(* PLC project CoDeSys External Library Template, WAGO e!COCKPIT e!COCKPIT, author 3S - Smart Software Solutions GmbH *)
(* stored: creationDateTime 2019-10-30T07:58:58.440898, version 3.5.5.30, modificationDateTime 2019-10-29T14:38:06.5373783, organization 3S - Smart Software Solutions GmbH *)
(* Library project template with all possible element types, docu and a sample project structure *)

TYPE alARRAYTablicaKomunikatow : ARRAY[1..2000] OF alSTRINGKomunikat;
END_TYPE

TYPE alARRAYTablicaKomunikatowDebug : ARRAY[1..100] OF typKomunikatDebug;
END_TYPE

TYPE alSTRINGjSON : STRING(10000);
END_TYPE

TYPE alSTRINGKomunikat : STRING(1024);
END_TYPE

{attribute 'qualified_only'}
{attribute 'strict'}
TYPE enumAlarmWartosc : (DUPA := 0, StanNormalny := 1, StanAlarmowy := 2);
END_TYPE

(* values of enumKlasaAlarmu: Bezpieczenstwa: najwyższy priorytet alarmu - alarm mogący mieć wpływ na bezpieczeństwo działania budynku; Krytyczny: wysoki priorytet alarmu - alarm istotny mogący doprowadzić do zaistnienia alarmu bezpieczeństwa; Ostrzezenie: średni priorytet alarmu - ostrzeżenie o nieprawidłowym działaniu któregoś z urządzeń; Informacyjny: niski priorytet alarm wyswietlany nie wymagajacy potwierdzenia; AwariaAutomatyki: alarm (podjrzenia) uszkodzenia lub nieprawidłowego działania automatyki; Wewnetrzny: alarm wewnetrzny niewyświetlany nie wymaga potwierdzenia; Systemowy: alarm systemowy niewyświetlany nie wymaga potwierdzenia *)

(* Nazwa bloku: Enumeracja - definicja klasy błędów Projekt: Bałtyckie Centrum Biznesu Budynek 2 Firma: Solwena Autor: Marcin Szumiło Aktualizacja: 2017-11-17-11:00-PK: aktualizacja względem pliku komunikacja 2019-02-13-14:56-AWy: dodanie klasy AwariaAutomatyki *)
{attribute 'qualified_only'}
{attribute 'strict'}
TYPE enumKlasaAlarmu : (Bezpieczenstwa := 0, Krytyczny := 1, Ostrzezenie := 2, Informacyjny := 3, AwariaAutomatyki := 8, Wewnetrzny := 9, Systemowy := 10);
END_TYPE

(* values of enumModbusKodyFunkcji: OdczytWyjscBitowych: odczyt stanu wyjść cyfrowych; OdczytWejscBitowych: odczyt stanu wejść cyfrowych; OdczytNRejestrow: odczyt dowolnej ilości rejestrów; OdczytNRejestrowWejsciowych: odczyt dowolnej ilości rejestrów wejściowych; ZapisBitu: zapis jednego bitu informacji; ZapisRejestru: zapis jednego rejestru; OdczytStatusu: odczyt statusu; ZapisNBitow: zapis dowolnej ilości bitów; ZapisNRejestrow: zapis dowolnej ilości rejestrów *)

(* Nazwa bloku: Enumeracja - definicja kodów funkcyjnych protokołu modbus Projekt: Bałtyckie Centrum Biznesu Budynek 2 Firma: Solwena Autor: Marcin Szumiło Wersja: 0.1.0.1 - 2017-01-10 *)
{attribute 'qualified_only'}
{attribute 'strict'}
TYPE enumModbusKodyFunkcji : (OdczytWyjscBitowych := 1, OdczytWejscBitowych := 2, OdczytNRejestrow := 3, OdczytNRejestrowWejsciowych := 4, ZapisBitu := 5, ZapisRejestru := 6, OdczytStatusu := 7, ZapisNBitow := 15, ZapisNRejestrow := 16);
END_TYPE

(* values of enumModbusStatus: BrakKomunikacji: problem z komunikacją; KomunikacjaPrawidlowa: komunikacja przebiegła prawidłowo *)

(* Nazwa bloku: Enumeracja - definicja kodów błędów w komunikacji modbus Projekt: Bałtyckie Centrum Biznesu Budynek 2 Firma: Solwena Autor: Marcin Szumiło Wersja: 0.1.0.1 - 2017-01-10 *)
{attribute 'qualified_only'}
{attribute 'strict'}
TYPE enumModbusStatus : (BrakKomunikacji := 1, KomunikacjaPrawidlowa := 2);
END_TYPE

(* values of enumPPPSAnalizatorDirisA40Error: BrakKomunikacji: brak komunikacji z analizatorem; BrakZmianyParametrow: alarm braku zmiany wartości paramterów (napięcie, prąd) *)

(* Autor: Paweł Kąkol, 2018-09-04-PK Prawa majątkowe: Solwena Sp. z o.o., Aktualizacje: 2019-02-18-AWy: alarm braku zmiany wartości napięcia lub prądu Opis: fb służy do obsługi alarmów w fb analizatora sieci ECA0 na budynkach PPP Sopot (ENGIE) Diris A40 *)
{attribute 'qualified_only'}
{attribute 'strict'}
TYPE enumPPPSAnalizatorDirisA40Error : (BrakKomunikacji := 1, BrakZmianyParametrow := 2);
END_TYPE

(* Autor: Paweł Kąkol, 2018-09-04-PK Prawa majątkowe: Solwena Sp. z o.o., Aktualizacje: 2019-02-18-AWy: alarm braku zmiany wartości napięcia lub prądu, zmiana klas alarmów Opis: fb służy do definicji klasy alarmów w fb analizatora sieci ECA0 na budynkach PPP Sopot (ENGIE) Diris A40 *)
{attribute 'qualified_only'}
{attribute 'strict'}
TYPE enumPPPSAnalizatorDirisA40ErrorKlasa : (BrakKomunikacji := enumKlasaAlarmu.AwariaAutomatyki, BrakZmianyParametrow := enumKlasaAlarmu.AwariaAutomatyki);
END_TYPE

(* values of enumPPPSBramkaSTC65RS485ModbusError: BrakKomunikacji: brak komunikacji (MODBUS RTU) z konwerterem; ResetKonwertera: reset konwertera; BrakTelegramowEnOcean: brak odbioru telegramów EnOcean (brak komunikacji EnOcean) *)

(* Autor: Paweł Kąkol, 2018-08-13-PK Prawa majątkowe: Solwena Sp. z o.o., Aktualizacje: 2018-09-10-PK - dodanie alarmów ResetKonwertera i BrakTelegramowEnOcean Opis: enum służy do obsługi alarmów w fb konwertera GTW0 na budynkach PPP Sopot *)
{attribute 'qualified_only'}
{attribute 'strict'}
TYPE enumPPPSBramkaSTC65RS485ModbusError : (BrakKomunikacji := 1, ResetKonwertera := 2, BrakTelegramowEnOcean := 3);
END_TYPE

(* Autor: Paweł Kąkol, 2018-08-13-PK Prawa majątkowe: Solwena Sp. z o.o., Aktualizacje: 2018-09-10-PK: dodanie klasy alarmów dla ResetKonwertera i BrakTelegramowEnOcean 2019-02-18-AWy: zmiana klas alarmów Opis: enum służy do definicji klas alarmów w fb konwertera GTW0 na budynkach PPP Sopot *)
{attribute 'qualified_only'}
{attribute 'strict'}
TYPE enumPPPSBramkaSTC65RS485ModbusErrorKlasa : (BrakKomunikacji := enumKlasaAlarmu.AwariaAutomatyki, ResetKonwertera := enumKlasaAlarmu.AwariaAutomatyki, BrakTelegramowEnOcean := enumKlasaAlarmu.AwariaAutomatyki);
END_TYPE

(* values of enumPPPSDestratyfikatorTBOXError: BrakKomunikacji: brak komunikacji z węzłem; AlarmCzujnika: alarm braku zmiany wartości czujnika temp. *)

(* Autor: Artur Wyszomirski, 2019-02-05-AWy Prawa majątkowe: Solwena Sp. z o.o., Aktualizacje: 2019-02-18-AWy - alarm czujnika temperatury Opis: enum służy do obsługi alarmów w fb węzła Frisko ATTOM1S na budynkach PPP Sopot (ENGIE) *)
{attribute 'qualified_only'}
{attribute 'strict'}
TYPE enumPPPSDestratyfikatorTBOXError : (BrakKomunikacji := 1, AlarmCzujnika := 2);
END_TYPE

(* Autor: Paweł Kąkol, 2018-09-03-PK Prawa majątkowe: Solwena Sp. z o.o., Aktualizacje: 2019-02-18-AWy: alarm czujnika temperatury 2019-02-18-AWy: zmiana klas alarmów Opis: enum służy do definicji klas alarmów w fb węzła Climatix POL63x na budynkach PPP Sopot (ENGIE) *)
{attribute 'qualified_only'}
{attribute 'strict'}
TYPE enumPPPSDestratyfikatorTBOXErrorKlasa : (BrakKomunikacji := enumKlasaAlarmu.AwariaAutomatyki, AlarmCzujnika := enumKlasaAlarmu.AwariaAutomatyki);
END_TYPE

(* values of enumPPPSFriskoATTOM1SError: BrakKomunikacji: brak komunikacji z węzłem; AlarmCzujnikaZewnetrznego: alarm braku zmiany wartości czujnika temp. zewnetrznj; AlarmCzujnikaZasilaniaObwoduCO: alarm braku zmiany wartości czujnika temp. zasilana obwod c. o.; BrakOsiagnieciaTemperaturyCO: alarm braku osiągnięcia temp. zadanej obwodu c. o.; BladIloscPomiarowTemperatury: alarm zbyt małej ilości pomiarów dokonanych w ciągu dnia do obliczenia średniej *)

(* Autor: Artur Wyszomirski, 2019-02-05-AWy Prawa majątkowe: Solwena Sp. z o.o., Aktualizacje: 2019-02-19-AWy: dodanie alarmów czujnika zew., zasilania c.o., braku osiągnięcia temperatury zadanej Opis: enum służy do obsługi alarmów w fb węzła Frisko ATTOM1S na budynkach PPP Sopot (ENGIE) *)
{attribute 'qualified_only'}
{attribute 'strict'}
TYPE enumPPPSFriskoATTOM1SError : (BrakKomunikacji := 1, AlarmCzujnikaZewnetrznego := 2, AlarmCzujnikaZasilaniaObwoduCO := 3, BrakOsiagnieciaTemperaturyCO := 4, BladIloscPomiarowTemperatury := 5);
END_TYPE

(* values of enumPPPSFriskoATTOM1SErrorKlasa: AlarmCzujnikaZewnetrznego: alarm braku zmiany wartości czujnika temp. zewnetrznj; AlarmCzujnikaZasilaniaObwoduCO: alarm braku zmiany wartości czujnika temp. zasilana obwod c. o.; BrakOsiagnieciaTemperaturyCO: alarm braku osiągnięcia temp. zadanej obwodu c. o.; BladIloscPomiarowTemperatury: alarm zbyt małej ilości pomiarów dokonanych w ciągu dnia do obliczenia średniej *)

(* Autor: Paweł Kąkol, 2018-09-03-PK Prawa majątkowe: Solwena Sp. z o.o., Aktualizacje: 2019-02-19-AWy: dodanie alarmów czujnika zew., zasilania c.o., braku osiągnięcia temperatury zadanej 2019-02-18-AWy: zmiana klas alarmów Opis: enum służy do definicji klas alarmów w fb węzła Climatix POL63x na budynkach PPP Sopot (ENGIE) *)
{attribute 'qualified_only'}
{attribute 'strict'}
TYPE enumPPPSFriskoATTOM1SErrorKlasa : (BrakKomunikacji := enumKlasaAlarmu.AwariaAutomatyki, AlarmCzujnikaZewnetrznego := enumKlasaAlarmu.AwariaAutomatyki, AlarmCzujnikaZasilaniaObwoduCO := enumKlasaAlarmu.AwariaAutomatyki, BrakOsiagnieciaTemperaturyCO := enumKlasaAlarmu.Ostrzezenie, BladIloscPomiarowTemperatury := enumKlasaAlarmu.AwariaAutomatyki);
END_TYPE

(* values of enumPPPSFriskoATTOM1STrybPracy: Zima: Zima; Lato: Lato; Auto: Automatyczny - przełączenie trybów uzależnione od temperatury zewnętrznej *)

(* Autor: Artur Wyszomirski, 22.05.2019 Prawa majątkowe: Solwena Sp. z o.o., Aktualizacje: Opis: enum służy do obsługi Trybów pracy fb węzła Frisko ATTO M1S na budynkach PPP Sopot (ENGIE) *)
{attribute 'qualified_only'}
{attribute 'strict'}
TYPE enumPPPSFriskoATTOM1STrybPracy : (Zima := 0, Lato := 1, Auto := 2);
END_TYPE

(* values of enumPPPSHarmonogramy: Ekonomiczny: Tryb pracy ekonomicznej; Komfort: Tryb pracy komfortu *)

(* Autor: Paweł Kąkol, 2018-09-10-PK Prawa majątkowe: Solwena Sp. z o.o., Aktualizacje: Opis: enum służy do obsługi Trybów pracy harmonogramu na budynkach PPP Sopot (ENGIE) *)
{attribute 'qualified_only'}
{attribute 'strict'}
TYPE enumPPPSHarmonogramy : (Ekonomiczny := 0, Komfort := 1);
END_TYPE

(* values of enumPPPSKlimatyzatorTroxSchoolairVError: BrakKomunikacji: brak komunikacji z węzłem; AlarmCzujnika: alarm braku zmiany wartości czujnika temp. *)

(* Autor: Artur Wyszomirski, 2019-02-05-AWy Prawa majątkowe: Solwena Sp. z o.o., Aktualizacje: 2019-02-18-AWy - alarm czujnika temperatury Opis: enum służy do obsługi alarmów w fb węzła Frisko ATTOM1S na budynkach PPP Sopot (ENGIE) *)
{attribute 'qualified_only'}
{attribute 'strict'}
TYPE enumPPPSKlimatyzatorTroxSchoolairVError : (BrakKomunikacji := 1, AlarmCzujnika := 2);
END_TYPE

(* Autor: Paweł Kąkol, 2018-09-03-PK Prawa majątkowe: Solwena Sp. z o.o., Aktualizacje: 2019-02-18-AWy: alarm czujnika temperatury 2019-02-18-AWy: zmiana klas alarmów Opis: enum służy do definicji klas alarmów w fb węzła Climatix POL63x na budynkach PPP Sopot (ENGIE) *)
{attribute 'qualified_only'}
{attribute 'strict'}
TYPE enumPPPSKlimatyzatorTroxSchoolairVErrorKlasa : (BrakKomunikacji := enumKlasaAlarmu.AwariaAutomatyki, AlarmCzujnika := enumKlasaAlarmu.AwariaAutomatyki);
END_TYPE

(* values of enumPPPSLicznikCieplaMultical403Error: BrakKomunikacji: Brak komunikacji z węzłem; AlarmCzujnikaPrzeplywu: Alarm braku zmiany wartości czujnika przepływu; AlarmCzujnikaZasilania: Alarm braku zmiany wartości czujnika temp. zasilania; AlarmCzujnikaPowrotu: Alarm braku zmiany wartości czujnika temp. powrotu *)

(* Autor: Artur Wyszomirski, 2019-08-07-AWy Prawa majątkowe: Solwena Sp. z o.o., Aktualizacje: Opis: Enumeracja alarmów w fb licznia ciepła Multical403 *)
{attribute 'qualified_only'}
{attribute 'strict'}
TYPE enumPPPSLicznikCieplaMultical403Error : (BrakKomunikacji := 1, AlarmCzujnikaPrzeplywu := 2, AlarmCzujnikaZasilania := 3, AlarmCzujnikaPowrotu := 4);
END_TYPE

(* values of enumPPPSLicznikCieplaMultical403ErrorKlasa: AlarmCzujnikaPrzeplywu: Alarm braku zmiany wartości czujnika przepływu; AlarmCzujnikaZasilania: Alarm braku zmiany wartości czujnika temp. zasilania; AlarmCzujnikaPowrotu: Alarm braku zmiany wartości czujnika temp. powrotu *)

(* Autor: Artur Wyszomirski, 2019-08-07-AWy Prawa majątkowe: Solwena Sp. z o.o., Aktualizacje: Opis: Klasy alarmów w fb licznia ciepła Multical403 *)
{attribute 'qualified_only'}
{attribute 'strict'}
TYPE enumPPPSLicznikCieplaMultical403ErrorKlasa : (BrakKomunikacji := enumKlasaAlarmu.AwariaAutomatyki, AlarmCzujnikaPrzeplywu := enumKlasaAlarmu.AwariaAutomatyki, AlarmCzujnikaZasilania := enumKlasaAlarmu.AwariaAutomatyki, AlarmCzujnikaPowrotu := enumKlasaAlarmu.Ostrzezenie);
END_TYPE

(* values of enumPPPSLicznikCieplaMultical602Error: BrakKomunikacji: Brak komunikacji z węzłem; AlarmCzujnikaPrzeplywu: Alarm braku zmiany wartości czujnika przepływu; AlarmCzujnikaZasilania: Alarm braku zmiany wartości czujnika temp. zasilania; AlarmCzujnikaPowrotu: Alarm braku zmiany wartości czujnika temp. powrotu *)

(* Autor: Artur Wyszomirski, 2019-08-08-AWy Prawa majątkowe: Solwena Sp. z o.o., Aktualizacje: Opis: Enumeracja alarmów w fb licznia ciepła Multical602 *)
{attribute 'qualified_only'}
{attribute 'strict'}
TYPE enumPPPSLicznikCieplaMultical602Error : (BrakKomunikacji := 1, AlarmCzujnikaPrzeplywu := 2, AlarmCzujnikaZasilania := 3, AlarmCzujnikaPowrotu := 4);
END_TYPE

(* values of enumPPPSLicznikCieplaMultical602ErrorKlasa: AlarmCzujnikaPrzeplywu: Alarm braku zmiany wartości czujnika przepływu; AlarmCzujnikaZasilania: Alarm braku zmiany wartości czujnika temp. zasilania; AlarmCzujnikaPowrotu: Alarm braku zmiany wartości czujnika temp. powrotu *)

(* Autor: Artur Wyszomirski, 2019-08-08-AWy Prawa majątkowe: Solwena Sp. z o.o., Aktualizacje: Opis: Klasy alarmów w fb licznia ciepła Multical602 *)
{attribute 'qualified_only'}
{attribute 'strict'}
TYPE enumPPPSLicznikCieplaMultical602ErrorKlasa : (BrakKomunikacji := enumKlasaAlarmu.AwariaAutomatyki, AlarmCzujnikaPrzeplywu := enumKlasaAlarmu.AwariaAutomatyki, AlarmCzujnikaZasilania := enumKlasaAlarmu.AwariaAutomatyki, AlarmCzujnikaPowrotu := enumKlasaAlarmu.Ostrzezenie);
END_TYPE

(* values of enumPPPSPomieszczenie: SalaLekcyjna: Sale lekcyjne, przedszkolne, świetlica, biblioteka (20 st. C); SalaNiemowlat: Sale niemowląt, dziecięce w żłobkach (24 st. C); Rehabilitacyjne: Pomieszczenia rehabilitacyjne SPON (24 st. C); Korytarz: Korytarze (20 st. C); Szatnia: Szatnie (16 st. C); SalaGimnastyczna: Sale gimnastyczne (16 st. C); Lazienka: Łazienki i ustępy (24 st. C); PomieszczenieBiurowe: Pomieszczenia biurowe i administracyjne (20 st. C); PomieszczenieMieszkalne: Pomieszczenia mieszkalne, przedpokoje, kuchnie (20 st. C); Magazyn: Pomieszczenia magazynowe (16 st. C) *)

(* Autor: Artur Wyszomirski, 2018-10-15-AW; Prawa majątkowe: Solwena Sp. z o.o., Aktualizacje: Opis: enum służy do obsługi rodzajów pomieszczeń w budynkach PPP Sopot (ENGIE) *)
{attribute 'qualified_only'}
{attribute 'strict'}
TYPE enumPPPSPomieszczenie : (SalaLekcyjna := 0, SalaNiemowlat := 1, Rehabilitacyjne := 2, Korytarz := 3, Szatnia := 4, SalaGimnastyczna := 5, Lazienka := 6, PomieszczenieBiurowe := 7, PomieszczenieMieszkalne := 8, Magazyn := 9);
END_TYPE

(* values of enumPPPSSilownikSABpError: BrakKomunikacji: brak komunikacji (po EnOcean) z siłownikiem; AlarmOgolny: alarm ogólny; DetekcjaOtwarciaOkna: błąd baterii; Defrost: defrost; AlarmCzujnika: alarm braku zmiany wartości czujnika temp. *)

(* Autor: Paweł Kąkol, 2018-09-04-PK Prawa majątkowe: Solwena Sp. z o.o., Aktualizacje: 2019-01-28-JC - defrost 2019-02-14-AWy - alarm czujnika temperatury Opis: enum służy do obsługi alarmów w fb siłownika (SAB+) HRU0 na budynkach PPP Sopot *)
{attribute 'qualified_only'}
{attribute 'strict'}
TYPE enumPPPSSilownikSABpError : (BrakKomunikacji := 1, AlarmOgolny := 2, DetekcjaOtwarciaOkna := 3, Defrost := 4, AlarmCzujnika := 5);
END_TYPE

(* Autor: Paweł Kąkol, 2018-09-04-PK Prawa majątkowe: Solwena Sp. z o.o., Aktualizacje: 2019-01-28-JC: defrost 2019-02-14-AWy: alarm czujnika temperatury 2019-02-18-AWy: zmiana klas alarmów Opis: enum służy do definicji klas alarmów w fb siłownika (SAB+) HRU0 na budynkach PPP Sopot *)
{attribute 'qualified_only'}
{attribute 'strict'}
TYPE enumPPPSSilownikSABpErrorKlasa : (BrakKomunikacji := enumKlasaAlarmu.AwariaAutomatyki, AlarmOgolny := enumKlasaAlarmu.Ostrzezenie, DetekcjaOtwarciaOkna := enumKlasaAlarmu.Informacyjny, Defrost := enumKlasaAlarmu.Bezpieczenstwa, AlarmCzujnika := enumKlasaAlarmu.AwariaAutomatyki);
END_TYPE

(* values of enumPPPSSilownikSABpServiceFlag: BrakDzialan: Brak rozkazu; TrybLetni: Rozkaz ustwienia trybu letniego; ZamkniecieZaworu: Rozkaz zamknięcia zaworu; OtwarcieZaworu: Rozkaz otwarcia zaworu; PozycjaGorna: Rozkaz pozycji górnej trzpienia (pozycja do transportu) - po jego uruchomieniu wymagana ponowna kalibracja; KalibracjaSilownika: Rozkaz uruchomienia sekwencji inicjalizacji siłownika *)

(* Autor: Paweł Kąkol, 2018-09-04-PK Prawa majątkowe: Solwena Sp. z o.o., Aktualizacje: Opis: enum służy do obsługi flagi serwisowej siłownika SAB+ (HRU0) na budynkach PPP Sopot (ENGIE) *)
{attribute 'qualified_only'}
{attribute 'strict'}
TYPE enumPPPSSilownikSABpServiceFlag : (BrakDzialan := 0, TrybLetni := 1, ZamkniecieZaworu := 2, OtwarcieZaworu := 3, PozycjaGorna := 4, KalibracjaSilownika := 5);
END_TYPE

(* values of enumPPPSSilownikTrybPracy: Manualny: Tryb pracy ręcznej; Automatyczny: Tryb pracy automatycznej *)

(* Autor: Artur Wyszomirski, 2018-09-25-AW Prawa majątkowe: Solwena Sp. z o.o., Aktualizacje: Opis: enum służy do obsługi Trybów pracy fb siłownika SABp (HRU0) na budynkach PPP Sopot (ENGIE) *)
{attribute 'qualified_only'}
{attribute 'strict'}
TYPE enumPPPSSilownikTrybPracy : (Manualny := 0, Automatyczny := 1);
END_TYPE

{attribute 'qualified_only'}
{attribute 'strict'}
TYPE enumPPPSUrzadenieStatus : (Nieaktywny := 1, Oczekiwanie := 2, Prawidlowy := 3, Ostrzezenie := 4, Awaria := 5, Krytyczny := 6);
END_TYPE

(* values of enumPPPSWezelClimatixPOL63xError: BrakKomunikacji: brak komunikacji z zadajnikiem; AlarmOgolnyBezpieczenstwa: alarm ogólny bezpieczeństwa; AlarmOgolnyKrytyczny: alarm ogólny krytyczny; AlarmOgolnyOstrzezenie: alarm ogólny ostrzeżenie; AlarmOgolnyInformacyjny: alarm ogólny informacyjny; AlarmCzujnikaZewnetrznego: alarm braku zmiany wartości czujnika temp. zewnetrznj; AlarmCzujnikaZasilaniaObwoduHC1: alarm braku zmiany wartości czujnika temp. zasilana obwodu HC1; AlarmCzujnikaZasilaniaObwoduDHW: alarm braku zmiany wartości czujnika temp. zasilana obwodu DHW; AlarmBrakuOsiagnieciaTemperaturyHC1: alarm braku osiągnięcia temp. zadanej obwodu HC1; AlarmBrakuOsiagnieciaTemperaturyDHW: alarm braku osiągnięcia temp. zadanej obwodu DHW; BladIloscPomiarowTemperatury: alarm zbyt małej ilości pomiarów dokonanych w ciągu dnia do obliczenia średniej *)

(* Autor: Paweł Kąkol, 2018-09-03-PK Prawa majątkowe: Solwena Sp. z o.o., Aktualizacje: 2019-02-14-AWy: dodanie alarmów czujników temp. zewnętrznej i zasilania obwodu HC1, DHW Opis: enum służy do obsługi alarmów w fb węzła Climatix POL63x na budynkach PPP Sopot (ENGIE) *)
{attribute 'qualified_only'}
{attribute 'strict'}
TYPE enumPPPSWezelClimatixPOL63xError : (BrakKomunikacji := 1, AlarmOgolnyBezpieczenstwa := 2, AlarmOgolnyKrytyczny := 3, AlarmOgolnyOstrzezenie := 4, AlarmOgolnyInformacyjny := 5, AlarmCzujnikaZewnetrznego := 6, AlarmCzujnikaZasilaniaObwoduHC1 := 7, AlarmCzujnikaZasilaniaObwoduDHW := 8, AlarmBrakuOsiagnieciaTemperaturyHC1 := 9, AlarmBrakuOsiagnieciaTemperaturyDHW := 10, BladIloscPomiarowTemperatury := 11);
END_TYPE

(* values of enumPPPSWezelClimatixPOL63xErrorKlasa: AlarmCzujnikaZewnetrznego: alarm braku zmiany wartości czujnika temp. zewnetrznj; AlarmCzujnikaZasilaniaObwoduHC1: alarm braku zmiany wartości czujnika temp. zasilana obwodu HC1; AlarmCzujnikaZasilaniaObwoduDHW: alarm braku zmiany wartości czujnika temp. zasilana obwodu DHW; AlarmBrakuOsiagnieciaTemperaturyHC1: alarm braku osiągnięcia temp. zadanej obwodu HC1; AlarmBrakuOsiagnieciaTemperaturyDHW: alarm braku osiągnięcia temp. zadanej obwodu DHW; BladIloscPomiarowTemperatury: alarm zbyt małej ilości pomiarów dokonanych w ciągu dnia do obliczenia średniej *)

(* Autor: Paweł Kąkol, 2018-09-03-PK Prawa majątkowe: Solwena Sp. z o.o., Aktualizacje: 2019-02-14-AWy: dodanie alarmów czujników temp. zewnętrznej i zasilania obwodu HC1, DHW 2019-02-18-AWy: zmiana klas alarmów Opis: enum służy do definicji klas alarmów w fb węzła Climatix POL63x na budynkach PPP Sopot (ENGIE) *)
{attribute 'qualified_only'}
{attribute 'strict'}
TYPE enumPPPSWezelClimatixPOL63xErrorKlasa : (BrakKomunikacji := enumKlasaAlarmu.AwariaAutomatyki, AlarmOgolnyBezpieczenstwa := enumKlasaAlarmu.Bezpieczenstwa, AlarmOgolnyKrytyczny := enumKlasaAlarmu.Krytyczny, AlarmOgolnyOstrzezenie := enumKlasaAlarmu.Ostrzezenie, AlarmOgolnyInformacyjny := enumKlasaAlarmu.Informacyjny, AlarmCzujnikaZewnetrznego := enumKlasaAlarmu.AwariaAutomatyki, AlarmCzujnikaZasilaniaObwoduHC1 := enumKlasaAlarmu.AwariaAutomatyki, AlarmCzujnikaZasilaniaObwoduDHW := enumKlasaAlarmu.AwariaAutomatyki, AlarmBrakuOsiagnieciaTemperaturyHC1 := enumKlasaAlarmu.Ostrzezenie, AlarmBrakuOsiagnieciaTemperaturyDHW := enumKlasaAlarmu.Ostrzezenie, BladIloscPomiarowTemperatury := enumKlasaAlarmu.AwariaAutomatyki);
END_TYPE

(* values of enumPPPSWezelClimatixPOL63xTrybPracy: Auto: Tryb pracy automatycznej; OchronaBudynku: Tryb utrzymania minimalnych nastaw dla ochrony budynku; Ekonomiczny: Tryb Ekonomiczny; Komfort: Tryb komfortu; ReczneWylaczenie: Ręczne, lokalne wyłączenie węzła *)

(* Autor: Paweł Kąkol, 2018-09-03-PK Prawa majątkowe: Solwena Sp. z o.o., Aktualizacje: Opis: enum służy do obsługi Trybów pracy fb węzła Climatix POL63x na budynkach PPP Sopot (ENGIE) *)
{attribute 'qualified_only'}
{attribute 'strict'}
TYPE enumPPPSWezelClimatixPOL63xTrybPracy : (Auto := 0, OchronaBudynku := 1, Ekonomiczny := 2, Komfort := 3, ReczneWylaczenie := 4);
END_TYPE

(* values of enumPPPSZadajnikError: BrakKomunikacji: brak komunikacji z zadajnikiem (po EnOcean); AlarmOgolny: alarm ogólny; AlarmCzujnika: alarm braku zmiany wartości czujnika temp. *)

(* Autor: Paweł Kąkol, 2018-08-13-PK Prawa majątkowe: Solwena Sp. z o.o., Aktualizacje: 2019-02-14-AWy - alarm czujnika temperatury Opis: enum służy do obsługi alarmów w fb zadajnika FCP0 na budynkach PPP Sopot *)
{attribute 'qualified_only'}
{attribute 'strict'}
TYPE enumPPPSZadajnikError : (BrakKomunikacji := 1, AlarmOgolny := 2, AlarmCzujnika := 3);
END_TYPE

(* Autor: Paweł Kąkol, 2018-08-13-PK Prawa majątkowe: Solwena Sp. z o.o., Aktualizacje: 2019-02-14-AWy: alarm czujnika temperatury 2019-02-18-AWy: zmiana klas alarmów Opis: enum służy do definicji klas alarmów w fb zadajnika FCP0 na budynkach PPP Sopot *)
{attribute 'qualified_only'}
{attribute 'strict'}
TYPE enumPPPSZadajnikErrorKlasa : (BrakKomunikacji := enumKlasaAlarmu.AwariaAutomatyki, AlarmOgolny := enumKlasaAlarmu.Ostrzezenie, AlarmCzujnika := enumKlasaAlarmu.AwariaAutomatyki);
END_TYPE

(* values of enumPPPSZadajnikTrybPracy: Manualny: Tryb pracy ręcznej; Automatyczny: Tryb pracy automatyczny *)

(* Autor: Paweł Kąkol, 2018-09-10-PK Prawa majątkowe: Solwena Sp. z o.o., Aktualizacje: 2018-10-02 - AW - Zmiana numeracji. Tryb Manualny na 0 2018-10-15 - AW - Zmiana numeracji. Dodanie trybów AutonomizacjaManualny i AutonomizacjaAutomatyczny 2018-12-12 - JB - Ujednolicenie trybów z siłownikiem SAB+. 2019-06-06 - AWy - Usunięcie trybów Wylaczenie, AutonomizacjaManualny i AutonomizacjaAutomatyczny oraz zmiana nazwy trybu Regulacja IZE na Automatyczny Opis: enum służy do obsługi Trybów pracy fb zadajnika SR04P (FCP0) na budynkach PPP Sopot (ENGIE) *)
{attribute 'qualified_only'}
{attribute 'strict'}
TYPE enumPPPSZadajnikTrybPracy : (Manualny := 0, Automatyczny := 1);
END_TYPE

{attribute 'qualified_only'}
{attribute 'strict'}
TYPE enumSystemError : (BrakHeartbetuzIZE := 1, NiezgodnaIloscKomunikatowOdebranychZIZE := 2, BladCRCWKomunikacieZIZE := 3, BladSzyfrowania := 4, ZaDuzaIloscKomunikatowWBuforze := 5, BladWalidacjiFullIdentifier := 6, BladFullIdentifierWHeartBeat := 7, BlokadaWysylaniaRamek := 8);
END_TYPE

{attribute 'qualified_only'}
{attribute 'strict'}
TYPE enumSystemErrorKlasa : (BrakHeartbetuzIZE := enumKlasaAlarmu.Krytyczny, NiezgodnaIloscKomunikatowOdebranychZIZE := enumKlasaAlarmu.Systemowy, BladCRCWKomunikacieZIZE := enumKlasaAlarmu.Systemowy, BladSzyfrowania := enumKlasaAlarmu.Systemowy, ZaDuzaIloscKomunikatowWBuforze := enumKlasaAlarmu.Systemowy, BladWalidacjiFullIdentifier := enumKlasaAlarmu.Systemowy, BladFullIdentifierWHeartBeat := enumKlasaAlarmu.Systemowy, BlokadaWysylaniaRamek := enumKlasaAlarmu.Systemowy);
END_TYPE

TYPE SILOWNIK_HRU : STRUCT
  sIdInstancji : STRING;
  intTrybPracy : INT;
  xBrakKomunikacjiIZE : BOOL;
  xBrakKomunikacjiPLC : BOOL;
  xPokazPanelHMI : BOOL := TRUE;
  rTemperaturaPomieszczenia : REAL;
  rNastawaPolozeniaSilownika : REAL;
  rZadanePolozenieSilownikaHMI : REAL;
  intTrybPracyHMI : INT := 1;
  xAutonomizacja : BOOL;
  xAlarmOgolny : BOOL;
  xBladBaterii : BOOL;
  xDetekcjaOtwarciaOkna : BOOL;
  sEnOceanIDodczytany : STRING;
  wCzasOdOstatniegoKomunikatu : WORD;
  xPoprawneParowanie : BOOL;
  xUczenieWlaczHMI : BOOL;
  xUczenieWlaczone : BOOL;
  xUsuwaniePotwierdzenieHMI : BOOL;
  xUsuwanieHMI : BOOL;
END_STRUCT;
END_TYPE

TYPE STEROWNIK_LAC : STRUCT
  xAutonomizacjaWyjscie : BOOL;
END_STRUCT;
END_TYPE

TYPE typHarmonogramDzien : STRUCT
  uintDzienTygodnia : UINT;
  arZdarzenia : ARRAY[0..24] OF typHarmonogramZdarzenie;
END_STRUCT;
END_TYPE

TYPE typHarmonogramJSON : STRUCT
  sPokoj : STRING(3);
  sPietro : STRING(2);
  arHarmonogramTygodniowy : ARRAY[0..6] OF typHarmonogramDzien;
  arWyjatki : ARRAY[0..24] OF typHarmonogramWyjatek;
END_STRUCT;
END_TYPE

TYPE typHarmonogramWyjatek : STRUCT
  dData : DATE;
  arZdarzenia : ARRAY[0..9] OF typHarmonogramZdarzenie;
END_STRUCT;
END_TYPE

TYPE typHarmonogramZdarzenie : STRUCT
  dtCzasRozpoczecia : DT;
  dtCzasZakonczenia : DT;
  sNazwaAtrybutu : STRING(15);
  sWartoscAtrybutu : STRING(15);
END_STRUCT;
END_TYPE

TYPE typKomunikat : STRUCT
  sZnacznik : STRING;
  sTypKomunikatu : STRING;
  sMnemonikWlasciciela : STRING;
  sMnemonikWlascicielaExt : STRING;
  sMACAdres : STRING;
  sIDZrodla : STRING;
  sIDZrodlaLokalizacja : STRING;
  sIDZrodlaUrzadzenie : STRING;
  sIDPrzeznaczenia : STRING;
  sIDPrzeznaczeniaLokalizacja : STRING;
  sIDPrzeznaczeniaUrzadzenie : STRING;
  sDlugoscPolaDanych : STRING;
  sMarkerCzasowy : STRING;
  sRezerwa : STRING;
  sDane : alSTRINGKomunikat;
END_STRUCT;
END_TYPE

TYPE typKomunikatDebug : STRUCT
  intGlobalnyZnacznikWysylkiUDP : INT;
  intGlobalnyZnacznikOdczytu : INT;
  intGlobalnyZnacznikZapisu : INT;
  intGlobalnaLiczbaKomunikatowWBuforze : INT;
  dtLokalnyCzasSterownika : DT;
  sDane : alSTRINGKomunikat;
END_STRUCT;
END_TYPE

TYPE typModbusOdczytCykliczny : STRUCT
  bAdresUrzadzenia : BYTE;  (* ID urządzenia SLAVE w sieci MODBUS *)
  bFunkcja : BYTE;  (* kod funkcji użytej w rozkazie MODBUS *)
  uiAdresRejestru : UINT;  (* rejestr startowy *)
  ltCzestotliwosc : LTIME;  (* po jakim czasie w ms ma być wysłany następny request *)
  ltZnacznikCzasuWyslania : LTIME;  (* znacznik czasowy próby wykonania rozkazu *)
  pZmiennaReferencyjna : POINTER TO WORD;  (* wskaźnik do zmiennej INT przechowującej wynik *)
END_STRUCT;
END_TYPE

TYPE typModbusOdczytZapisZadanie : STRUCT
  bAdresUrzadzenia : BYTE;  (* ID urządzenia SLAVE w sieci MODBUS *)
  bFunkcja : BYTE;  (* kod funkcji użytej w rozkazie MODBUS *)
  uiAdresRejestru : UINT;  (* rejestr startowy *)
  pZmiennaDoOdczytu : POINTER TO WORD;  (* wskaźnik do zmiennej INT przechowującej wynik *)
  wWartoscDoZapisania : WORD;  (* wartość do zapisania *)
END_STRUCT;
END_TYPE

TYPE typModbusRTUParametryKomunikacji : STRUCT
  xKomunikacjaAktywna : BOOL;
  typNazwaPortuKomunikacyjnego : WagoTypesCom.I_WagoSysComBase;
  udiPredkosc : UDINT;
  usiBityDanych : USINT;
  eParzystosc : eTTYParity;
  eBityStopu : eTTYStopBits;
  eHandshake : eTTYHandshake;
  eDuplex : eTTYPhysicalLayer;
  eTypRamki : eMbFrameType;
  tTimeout : TIME;
END_STRUCT;
END_TYPE

TYPE typModbusTCPParametryKomunikacji : STRUCT
  xKomunikacjaAktywna : BOOL;
  sAdresTCP : STRING;
  wPortTCP : WORD;
  utPodtrzymajWtyczkeTCP : typKeepAlive;
  eTypRamki : eMbFrameType;
  tTimeOut : TIME;
END_STRUCT;
END_TYPE

TYPE typWirtualnePomieszczenie : STRUCT
  sIDPomieszczenia : STRING;
  intObecnosc : INT := -1;
END_STRUCT;
END_TYPE

TYPE ZADAJNIK_FCP : STRUCT
  sIdInstancji : STRING;
  rTemperaturaNastawiona : REAL;
  rTemperaturaPomieszczenia : REAL;
  rTemperaturaBazowaHMI : REAL := 293.15;
  rSkalaPotencjometruAutonomizacja : REAL := 1;
  rTemperaturaBazowaAutoAutonomizacja : REAL := 293.15;
  intTrybPracy : INT;
  xBrakKomunikacjiIZE : BOOL;
  xBrakKomunikacjiPLC : BOOL;
  xPokazPanelHMI : BOOL := TRUE;
  intTrybPracyHMI : INT := 1;
  xAutonomizacja : BOOL;
  sEnOceanIDodczytany : STRING;
  wCzasOdOstatniegoKomunikatu : WORD;
  xZwiekszTemperature : BOOL;
  xZmniejszTemperature : BOOL;
END_STRUCT;
END_TYPE

(* Nazwa bloku: Blok funkcyjny konwersji liczby decymalnej na binarną Autor: Jan Bartczak Wersja: v1.0.0 - 2018-06-22 *)
FUNCTION_BLOCK fbDecToBin
  VAR_INPUT
    wWordWejsciowy : WORD;
    intIloscBitow : INT;
  END_VAR
  VAR_OUTPUT
    arBity : ARRAY[0..16] OF BYTE;
  END_VAR
  VAR
    intWejsciowy : UINT;
    bBajtPojedynczy : BYTE;
    intWord : WORD;
    intI : INT;
  END_VAR

            intWejsciowy := WORD_TO_UINT(wWordWejsciowy);
intIloscBitow := intIloscBitow - 1;
FOR intI := 0 TO intIloscBitow BY 1 DO
	intWord := (intWejsciowy MOD 2);
	bBajtPojedynczy := UINT_TO_BYTE(intWord);
	arBity[intI] := bBajtPojedynczy;
	intWejsciowy := intWejsciowy/2;
END_FOR;

          
END_FUNCTION_BLOCK

FUNCTION_BLOCK fbFiltrWartoscAnalogowa
  VAR_INPUT
    rWartoscWejsciowa : REAL;
    rWartoscWejsciowaZaraportowana : REAL;
    rDeadband : REAL;
    tCzasMinimalny : TIME := TIME#5s0ms;
    tCzasMaksymalny : TIME := TIME#1m0s0ms;
    rWynikMnoznik : REAL := 1;
    rWynikOffset : REAL := 0;
  END_VAR
  VAR_OUTPUT
    rWartoscWyjsciowa : REAL;
  END_VAR
  VAR
    rWartoscWejsciowaZaraportowanaReferencja : REAL;
    fbCzasMinimalny : TON;
    fbCzasMaksymalny : TON;
    xCzasMinimalny : BOOL;
    xCzasMaksymalny : BOOL;
  END_VAR

            xCzasMinimalny := TRUE;
xCzasMaksymalny := TRUE;	

IF rWartoscWejsciowaZaraportowana <> rWartoscWejsciowaZaraportowanaReferencja THEN
	rWartoscWejsciowaZaraportowanaReferencja := rWartoscWejsciowaZaraportowana;
	xCzasMinimalny := FALSE;
	xCzasMaksymalny := FALSE;	
END_IF

IF fbCzasMinimalny.Q AND ABS(rWartoscWyjsciowa - (rWartoscWejsciowa * rWynikMnoznik + rWynikOffset)) > rDeadband THEN
	rWartoscWyjsciowa := rWartoscWejsciowa * rWynikMnoznik + rWynikOffset;
	xCzasMinimalny := FALSE;
	xCzasMaksymalny := FALSE;
END_IF

IF fbCzasMaksymalny.Q AND rWartoscWyjsciowa <> rWartoscWejsciowa * rWynikMnoznik + rWynikOffset THEN
	rWartoscWyjsciowa := rWartoscWejsciowa * rWynikMnoznik + rWynikOffset;
	xCzasMinimalny := FALSE;
	xCzasMaksymalny := FALSE;
END_IF

fbCzasMinimalny(IN := xCzasMinimalny, PT := tCzasMinimalny);
fbCzasMaksymalny(IN := xCzasMaksymalny , PT := tCzasMaksymalny);
          
END_FUNCTION_BLOCK

FUNCTION_BLOCK fbModbusDriverRTU
  VAR_INPUT
    intOdczytZapisZadanieRozmiarBufora : INT;
    arRTUParametryKomunikacji : ARRAY[1..256] OF typModbusRTUParametryKomunikacji;
  END_VAR
  VAR_IN_OUT
    arOdczytCykliczny : ARRAY[1..5000] OF typModbusOdczytCykliczny;
    arOdczytZapisZadanie : ARRAY[1..1000] OF typModbusOdczytZapisZadanie;
    arStatusKomunikacji : ARRAY[1..256] OF INT;
    intZnacznikOdczytuZapisuZadanie : INT;
  END_VAR
  VAR
    ModbusMasterRTU : FbMbMasterSerial;
    arRTUParametryKomunikacjiPoprz : ARRAY[1..256] OF typModbusRTUParametryKomunikacji;
    utZapytanie : typMBQuery;
    utZapytaniePoprz : typMBQuery;
    utOdpowiedz : typMbResponse;
    xStatusPolaczenia : BOOL;
    xBladKomunikacji : BOOL;
    typStatusKomunikacji : WagoSysErrorBase.FbResult;
    tCzasPonowienia : LTIME := LTIME#15s0ms0us0ns;
    tCzasStabilnosciKomunikacji : LTIME := LTIME#30s0ms0us0ns;  (* czas po jakim driver raportuje poprawną komunikację po jej faktycznym odzyskaniu - czas powinien być większy niż czas tCzasPonawiania *)
    xDriverWykonajKomunikacje : BOOL;  (* zmienna sygnalizujaca konicznosc wykonania zapisu/odczytu do Modbus RTU *)
    tonDriverWykonajKomunikacje : TON;  (* Opóżnienie włączenia triggera wysłania komunikatu po włączeniu drivera MODBUSa *)
    xDriverWykonajKomunikacjeTrigger : BOOL;  (* Trigger wysłania komunikatu MODBUS *)
    ftrigDriverWykonajKomunikacjeTrigger : F_TRIG;  (* Zbocze opadające triggera wysłania komunikatu *)
    arStatusKomunikacjiTimestampOstatniaProba : ARRAY[1..256] OF LTIME;
    arStatusKomunikacjiTimestampOstatniBlad : ARRAY[1..256] OF LTIME;
    negWykonaj : F_TRIG;
    intZnacznikDriveraOdczytuCyklicznego : INT := 0;
    intZnacznikDriveraOdczytuZapisuZadanie : INT := 0;
    intZnacznikOdczytuCyklicznegoReferencja : INT;
    intZnacznikOdczytuCyklicznegoPoczatek : INT;
    intZnacznikOdczytuZapisuZadanieReferencja : INT;
    intZnacznikPomocniczy : INT;
    intOdczytZadanieTablica : INT;
    intOdczytCyklicznyTablica : INT;
    intOdczytCyklicznyTablicaIlosc : INT;
    intLoop : INT;
    intLoopOverflow : INT;
    statusbledu : WagoSysErrorBase.FbResult;
    jakiezapytanie : typMBQuery;
    intDebugZnacznik : INT;  (* debug *)
    arDebugZapytanie : ARRAY[0..5000] OF typMBQuery;
    arDebugOdpowiedz : ARRAY[0..5000] OF typMbResponse;
    typDebugOdczytZapisZadanie : ARRAY[0..5000] OF typModbusOdczytZapisZadanie;
    arDebugCzas : ARRAY[0..5000] OF DT;
    inttest : DINT;
    ctuLicznikBledow : CTU;  (* Licznik błędów *)
  END_VAR

            (*			
Autor:					N/A
Prawa majątkowe: 		Solwena Sp. z o.o., 
Aktualizacje:								

Opis:					Obsługa komunikacji MODBUS
						
Aktualizacje:			2019-09-13-AWy: zmiana sposobu uruchamiania drivera MODBUSowego ModbusMasterRTU i wysyłania komunkatów.
						2019-10-18-AWy: dodanie licznika błędów
						2019-10-22-AWy: zmiana opóżnienia włączenia drivera po zakończeniu komunikacji
						
Rozwój:					Możliwe jest przyspieszenie drivera poprzez nie restartowanie po każdej komunikacji a jedynie wtedy, gdy ulegną zmianie parametry komunikacji.						
	
*)

// obsługa odczytu/zapisu danych na żądanie

IF intZnacznikDriveraOdczytuZapisuZadanie <> intZnacznikOdczytuZapisuZadanie AND NOT xDriverWykonajKomunikacje THEN
	fnTablicaKomunikatowInkrementacja(intRozmiarTablicy := intOdczytZapisZadanieRozmiarBufora, intWskaznik := intZnacznikDriveraOdczytuZapisuZadanie);
	IF arStatusKomunikacji[arOdczytZapisZadanie[intZnacznikDriveraOdczytuZapisuZadanie].bAdresUrzadzenia] = enumModbusStatus.KomunikacjaPrawidlowa THEN
		xDriverWykonajKomunikacje := TRUE;
		utZapytanie.bUnitId := arOdczytZapisZadanie[intZnacznikDriveraOdczytuZapisuZadanie].bAdresUrzadzenia;
		utZapytanie.bFunctionCode := arOdczytZapisZadanie[intZnacznikDriveraOdczytuZapisuZadanie].bFunkcja;
		utZapytanie.uiReadQuantity := 1;
		utZapytanie.uiReadAddress := arOdczytZapisZadanie[intZnacznikDriveraOdczytuZapisuZadanie].uiAdresRejestru;
		utZapytanie.uiWriteAddress := arOdczytZapisZadanie[intZnacznikDriveraOdczytuZapisuZadanie].uiAdresRejestru;
		utZapytanie.awWriteData[0] := arOdczytZapisZadanie[intZnacznikDriveraOdczytuZapisuZadanie].wWartoscDoZapisania;
		utZapytanie.uiWriteQuantity := 1;
		intOdczytZadanieTablica := intZnacznikDriveraOdczytuZapisuZadanie;
	END_IF
END_IF

// obsługa odczytu cyklicznego zmiennych zapisanych w tabeli

IF NOT xDriverWykonajKomunikacje THEN 
	
	intZnacznikOdczytuCyklicznegoReferencja := intZnacznikDriveraOdczytuCyklicznego;
	intZnacznikDriveraOdczytuCyklicznego := intZnacznikDriveraOdczytuCyklicznego + 1;
	IF arOdczytCykliczny[intZnacznikDriveraOdczytuCyklicznego].bAdresUrzadzenia = 0 THEN
		intZnacznikDriveraOdczytuCyklicznego := 1;
	END_IF

	WHILE intZnacznikOdczytuCyklicznegoReferencja <> intZnacznikDriveraOdczytuCyklicznego AND _GetLongTime() - arStatusKomunikacjiTimestampOstatniaProba[arOdczytCykliczny[intZnacznikDriveraOdczytuCyklicznego].bAdresUrzadzenia] < tCzasPonowienia AND
			_GetLongTime() - arOdczytCykliczny[intZnacznikDriveraOdczytuCyklicznego].ltZnacznikCzasuWyslania < arOdczytCykliczny[intZnacznikDriveraOdczytuCyklicznego].ltCzestotliwosc DO
		intZnacznikDriveraOdczytuCyklicznego := intZnacznikDriveraOdczytuCyklicznego + 1;
		IF arOdczytCykliczny[intZnacznikDriveraOdczytuCyklicznego].bAdresUrzadzenia = 0 THEN
			intZnacznikDriveraOdczytuCyklicznego := 1;
		END_IF
	END_WHILE

// zapis adresu startowego rejestrów do zapisu

	IF intZnacznikOdczytuCyklicznegoReferencja <> intZnacznikDriveraOdczytuCyklicznego THEN
		xDriverWykonajKomunikacje := TRUE;
		arStatusKomunikacjiTimestampOstatniaProba[arOdczytCykliczny[intZnacznikDriveraOdczytuCyklicznego].bAdresUrzadzenia] := _GetLongTime();
		utZapytanie.bUnitId := arOdczytCykliczny[intZnacznikDriveraOdczytuCyklicznego].bAdresUrzadzenia;
		utZapytanie.bFunctionCode := arOdczytCykliczny[intZnacznikDriveraOdczytuCyklicznego].bFunkcja;
		utZapytanie.uiReadAddress := arOdczytCykliczny[intZnacznikDriveraOdczytuCyklicznego].uiAdresRejestru;
		utZapytanie.uiReadQuantity := 1;
		intOdczytCyklicznyTablica := intZnacznikDriveraOdczytuCyklicznego;
		intZnacznikOdczytuCyklicznegoReferencja := intZnacznikDriveraOdczytuCyklicznego;
		intZnacznikPomocniczy := intZnacznikDriveraOdczytuCyklicznego + 1;
		IF arOdczytCykliczny[intZnacznikPomocniczy].bAdresUrzadzenia = 0 THEN
			intZnacznikPomocniczy := 1;
		END_IF

// sprawdzenie czy następne żądanie nie jest w kolejności do bieżącego jeśli tak to grupuje je w jedno zapytanie

		WHILE (arOdczytCykliczny[intZnacznikPomocniczy].uiAdresRejestru - arOdczytCykliczny[intZnacznikDriveraOdczytuCyklicznego].uiAdresRejestru = 1 AND
				arOdczytCykliczny[intZnacznikPomocniczy].bFunkcja = arOdczytCykliczny[intZnacznikDriveraOdczytuCyklicznego].bFunkcja AND
				arOdczytCykliczny[intZnacznikPomocniczy].bAdresUrzadzenia = arOdczytCykliczny[intZnacznikDriveraOdczytuCyklicznego].bAdresUrzadzenia) DO
				
			utZapytanie.uiReadQuantity := utZapytanie.uiReadQuantity + 1;
			intZnacznikDriveraOdczytuCyklicznego := intZnacznikDriveraOdczytuCyklicznego + 1;
			IF arOdczytCykliczny[intZnacznikDriveraOdczytuCyklicznego].bAdresUrzadzenia = 0 THEN
				intZnacznikDriveraOdczytuCyklicznego := 1;
			END_IF
			intZnacznikPomocniczy := intZnacznikDriveraOdczytuCyklicznego + 1;
			IF arOdczytCykliczny[intZnacznikPomocniczy].bAdresUrzadzenia = 0 THEN
				intZnacznikPomocniczy := 1;
			END_IF
		END_WHILE
		intOdczytCyklicznyTablicaIlosc := UINT_TO_INT(utZapytanie.uiReadQuantity);
	END_IF
END_IF

// driver komunikacyjny MODBUS RTU
	// Na potrzeby obsługi komunikacji w kilku prędkościach: ModbusMasterRTU jest włączany (xConnect := TRUE), wprowadzane są nowe parametry komunikacji, a następnie triggerowane jest wysłanie komunikatu
	// (xTrigger := TRUE). Następnie ModbusMasterRTU jest wyłączany (xConnect := FALSE) i algorytm zaczyna się od nowa.

ftrigDriverWykonajKomunikacjeTrigger(CLK := xDriverWykonajKomunikacjeTrigger);
IF ftrigDriverWykonajKomunikacjeTrigger.Q THEN
	xDriverWykonajKomunikacje := FALSE;
END_IF

tonDriverWykonajKomunikacje(IN := xDriverWykonajKomunikacje, PT := T#1000MS); // Opóżnienie konieczne ze względu na nieprawidłowe działanie drivera przy zbyt szybkim wysyłaniu komunikatu po włączeniu drivera
IF tonDriverWykonajKomunikacje.Q THEN
	xDriverWykonajKomunikacjeTrigger := TRUE;
END_IF		

ModbusMasterRTU(xConnect := 		xDriverWykonajKomunikacje,
				I_Port := 			arRTUParametryKomunikacji[utZapytanie.bUnitId].typNazwaPortuKomunikacyjnego , 
				eFrameType := 		arRTUParametryKomunikacji[utZapytanie.bUnitId].eTypRamki , 
				udiBaudrate := 		arRTUParametryKomunikacji[utZapytanie.bUnitId].udiPredkosc , 
				usiDataBits := 		arRTUParametryKomunikacji[utZapytanie.bUnitId].usiBityDanych , 
				eParity := 			arRTUParametryKomunikacji[utZapytanie.bUnitId].eParzystosc , 
				eStopBits := 		arRTUParametryKomunikacji[utZapytanie.bUnitId].eBityStopu , 
				eHandshake :=		arRTUParametryKomunikacji[utZapytanie.bUnitId].eHandshake , 
				ePhysical := 		arRTUParametryKomunikacji[utZapytanie.bUnitId].eDuplex , 
				tTimeOut := 		arRTUParametryKomunikacji[utZapytanie.bUnitId].tTimeout , 
 
				xTrigger := 		xDriverWykonajKomunikacjeTrigger , 
				utQuery := 			utZapytanie , 
				utResponse := 		utOdpowiedz ,
 
				xError => 			xBladKomunikacji);
				
// Licznik błędów
ctuLicznikBledow(CU := ModbusMasterRTU.xError, PV := 65535);
	
// obługa akcji po zakończeniu zadania komunikacji (zapis wartości , zapis błędu itd)
	
negWykonaj(CLK := xDriverWykonajKomunikacjeTrigger);

IF negWykonaj.Q THEN
// jeżeli był błąd komunikacji wpisz go do tablicy błędów

	IF xBladKomunikacji THEN
		arStatusKomunikacji[utZapytanie.bUnitId] := enumModbusStatus.BrakKomunikacji;
		statusbledu := ModbusMasterRTU.oStatus;
		jakiezapytanie := utZapytanie;
		arStatusKomunikacjiTimestampOstatniBlad[utZapytanie.bUnitId] := _GetLongTime();
		IF utZapytaniePoprz.bFunctionCode = 0 THEN
			utZapytaniePoprz := utZapytanie;
		END_IF
		IF arRTUParametryKomunikacjiPoprz[3].udiPredkosc = 0 THEN
			arRTUParametryKomunikacjiPoprz := arRTUParametryKomunikacji;
		END_IF
	ELSE
		IF _GetLongTime() - arStatusKomunikacjiTimestampOstatniBlad[utZapytanie.bUnitId] > tCzasStabilnosciKomunikacji AND arStatusKomunikacji[utZapytanie.bUnitId] <> enumModbusStatus.KomunikacjaPrawidlowa THEN	
			arStatusKomunikacji[utZapytanie.bUnitId] := enumModbusStatus.KomunikacjaPrawidlowa;
		END_IF

// jeżeli zapytanie było żądaniem  wysłania danych

		IF utZapytanie.bFunctionCode = enumModbusKodyFunkcji.OdczytWejscBitowych OR utZapytanie.bFunctionCode = enumModbusKodyFunkcji.OdczytWyjscBitowych OR
			utZapytanie.bFunctionCode = enumModbusKodyFunkcji.OdczytNRejestrow OR utZapytanie.bFunctionCode = enumModbusKodyFunkcji.OdczytNRejestrowWejsciowych THEN
			intZnacznikOdczytuCyklicznegoPoczatek := 0;
		
// jeżeli był wykonany rozkaz odczytu danych z cyklu "na żądanie" - DOŁOŻONO KAWAŁEK KODU DEBUGUJĄCEGO - ZATRZYMYWANIE SIĘ STEROWNIKA NA ZAREMOWANEJ LINII

			IF intOdczytZadanieTablica <> 0 THEN
				arDebugZapytanie[intDebugZnacznik] := utZapytanie;
				arDebugOdpowiedz[intDebugZnacznik] := utOdpowiedz;
				typDebugOdczytZapisZadanie[intDebugZnacznik] := arOdczytZapisZadanie[intZnacznikDriveraOdczytuZapisuZadanie];				
				arDebugCzas[intDebugZnacznik] := FuGetDateAndTime();
				fnTablicaKomunikatowInkrementacja(intRozmiarTablicy := 900, intWskaznik := intDebugZnacznik);
//				arOdczytZapisZadanie[intZnacznikDriveraOdczytuZapisuZadanie].pZmiennaDoOdczytu^ := utOdpowiedz.awData[0];
			END_IF

// jeżeli był wykonany rozkaz odczytu danych z cyklu "cykliczny"

			IF intOdczytCyklicznyTablica <> 0 THEN
				intLoopOverflow:=1;
				FOR intLoop := 1 TO intOdczytCyklicznyTablicaIlosc DO
					IF arOdczytCykliczny[intOdczytCyklicznyTablica + intLoop - 1].pZmiennaReferencyjna <> null THEN
					arOdczytCykliczny[intOdczytCyklicznyTablica + intLoop - 1].pZmiennaReferencyjna^ := utOdpowiedz.awData[intLoop - 1];
					arOdczytCykliczny[intOdczytCyklicznyTablica + intLoop - 1].ltZnacznikCzasuWyslania := _GetLongTime();
					ELSE
					arOdczytCykliczny[intLoopOverflow].pZmiennaReferencyjna^ := utOdpowiedz.awData[intLoop - 1];
					arOdczytCykliczny[intLoopOverflow].ltZnacznikCzasuWyslania := _GetLongTime();
					intLoopOverflow:=intLoopOverflow+1;
					END_IF
				END_FOR
			END_IF
		END_IF
	END_IF
	intOdczytZadanieTablica := 0;
	intOdczytCyklicznyTablica := 0;
	intOdczytCyklicznyTablicaIlosc := 0;
END_IF


          
END_FUNCTION_BLOCK

FUNCTION_BLOCK fbModbusDriverRTUStary
  VAR_INPUT
    intOdczytZapisZadanieRozmiarBufora : INT;
    arRTUParametryKomunikacji : ARRAY[1..256] OF typModbusRTUParametryKomunikacji;
  END_VAR
  VAR_IN_OUT
    arOdczytCykliczny : ARRAY[1..5000] OF typModbusOdczytCykliczny;
    arOdczytZapisZadanie : ARRAY[1..1000] OF typModbusOdczytZapisZadanie;
    arStatusKomunikacji : ARRAY[1..256] OF INT;
    intZnacznikOdczytuZapisuZadanie : INT;
  END_VAR
  VAR
    ModbusMasterRTU : FbMbMasterSerial;
    arRTUParametryKomunikacjiPoprz : ARRAY[1..256] OF typModbusRTUParametryKomunikacji;
    utZapytanie : typMBQuery;
    utZapytaniePoprz : typMBQuery;
    utOdpowiedz : typMbResponse;
    xStatusPolaczenia : BOOL;
    xBladKomunikacji : BOOL;
    typStatusKomunikacji : WagoSysErrorBase.FbResult;
    tCzasPonowienia : LTIME := LTIME#15s0ms0us0ns;
    tCzasStabilnosciKomunikacji : LTIME := LTIME#30s0ms0us0ns;  (* czas po jakim driver raportuje poprawną komunikację po jej faktycznym odzyskaniu - czas powinien być większy niż czas tCzasPonawiania *)
    xDriverWykonajKomunikacje : BOOL;  (* zmienna sygnalizujaca konicznosc wykonania zapisu/odczytu do Modbus RTU *)
    arStatusKomunikacjiTimestampOstatniaProba : ARRAY[1..256] OF LTIME;
    arStatusKomunikacjiTimestampOstatniBlad : ARRAY[1..256] OF LTIME;
    negWykonaj : F_TRIG;
    intZnacznikDriveraOdczytuCyklicznego : INT := 0;
    intZnacznikDriveraOdczytuZapisuZadanie : INT := 0;
    intZnacznikOdczytuCyklicznegoReferencja : INT;
    intZnacznikOdczytuCyklicznegoPoczatek : INT;
    intZnacznikOdczytuZapisuZadanieReferencja : INT;
    intZnacznikPomocniczy : INT;
    intOdczytZadanieTablica : INT;
    intOdczytCyklicznyTablica : INT;
    intOdczytCyklicznyTablicaIlosc : INT;
    intLoop : INT;
    intLoopOverflow : INT;
    statusbledu : WagoSysErrorBase.FbResult;
    jakiezapytanie : typMBQuery;
    intDebugZnacznik : INT;  (* debug *)
    arDebugZapytanie : ARRAY[0..5000] OF typMBQuery;
    arDebugOdpowiedz : ARRAY[0..5000] OF typMbResponse;
    typDebugOdczytZapisZadanie : ARRAY[0..5000] OF typModbusOdczytZapisZadanie;
    arDebugCzas : ARRAY[0..5000] OF DT;
    inttest : DINT;
  END_VAR

            // obsługa odczytu/zapisu danych na żądanie

IF intZnacznikDriveraOdczytuZapisuZadanie <> intZnacznikOdczytuZapisuZadanie AND NOT xDriverWykonajKomunikacje THEN
	fnTablicaKomunikatowInkrementacja(intRozmiarTablicy := intOdczytZapisZadanieRozmiarBufora, intWskaznik := intZnacznikDriveraOdczytuZapisuZadanie);
	IF arStatusKomunikacji[arOdczytZapisZadanie[intZnacznikDriveraOdczytuZapisuZadanie].bAdresUrzadzenia] = enumModbusStatus.KomunikacjaPrawidlowa THEN
		xDriverWykonajKomunikacje := TRUE;
		utZapytanie.bUnitId := arOdczytZapisZadanie[intZnacznikDriveraOdczytuZapisuZadanie].bAdresUrzadzenia;
		utZapytanie.bFunctionCode := arOdczytZapisZadanie[intZnacznikDriveraOdczytuZapisuZadanie].bFunkcja;
		utZapytanie.uiReadQuantity := 1;
		utZapytanie.uiReadAddress := arOdczytZapisZadanie[intZnacznikDriveraOdczytuZapisuZadanie].uiAdresRejestru;
		utZapytanie.uiWriteAddress := arOdczytZapisZadanie[intZnacznikDriveraOdczytuZapisuZadanie].uiAdresRejestru;
		utZapytanie.awWriteData[0] := arOdczytZapisZadanie[intZnacznikDriveraOdczytuZapisuZadanie].wWartoscDoZapisania;
		utZapytanie.uiWriteQuantity := 1;
		intOdczytZadanieTablica := intZnacznikDriveraOdczytuZapisuZadanie;
	END_IF
END_IF

// obsługa odczytu cyklicznego zmiennych zapisanych w tabeli

IF NOT xDriverWykonajKomunikacje THEN 
	
	intZnacznikOdczytuCyklicznegoReferencja := intZnacznikDriveraOdczytuCyklicznego;
	intZnacznikDriveraOdczytuCyklicznego := intZnacznikDriveraOdczytuCyklicznego + 1;
	IF arOdczytCykliczny[intZnacznikDriveraOdczytuCyklicznego].bAdresUrzadzenia = 0 THEN
		intZnacznikDriveraOdczytuCyklicznego := 1;
	END_IF

	WHILE intZnacznikOdczytuCyklicznegoReferencja <> intZnacznikDriveraOdczytuCyklicznego AND _GetLongTime() - arStatusKomunikacjiTimestampOstatniaProba[arOdczytCykliczny[intZnacznikDriveraOdczytuCyklicznego].bAdresUrzadzenia] < tCzasPonowienia AND
			_GetLongTime() - arOdczytCykliczny[intZnacznikDriveraOdczytuCyklicznego].ltZnacznikCzasuWyslania < arOdczytCykliczny[intZnacznikDriveraOdczytuCyklicznego].ltCzestotliwosc DO
		intZnacznikDriveraOdczytuCyklicznego := intZnacznikDriveraOdczytuCyklicznego + 1;
		IF arOdczytCykliczny[intZnacznikDriveraOdczytuCyklicznego].bAdresUrzadzenia = 0 THEN
			intZnacznikDriveraOdczytuCyklicznego := 1;
		END_IF
	END_WHILE

// zapis adresu startowego rejestrów do zapisu

	IF intZnacznikOdczytuCyklicznegoReferencja <> intZnacznikDriveraOdczytuCyklicznego THEN
		xDriverWykonajKomunikacje := TRUE;
		arStatusKomunikacjiTimestampOstatniaProba[arOdczytCykliczny[intZnacznikDriveraOdczytuCyklicznego].bAdresUrzadzenia] := _GetLongTime();
		utZapytanie.bUnitId := arOdczytCykliczny[intZnacznikDriveraOdczytuCyklicznego].bAdresUrzadzenia;
		utZapytanie.bFunctionCode := arOdczytCykliczny[intZnacznikDriveraOdczytuCyklicznego].bFunkcja;
		utZapytanie.uiReadAddress := arOdczytCykliczny[intZnacznikDriveraOdczytuCyklicznego].uiAdresRejestru;
		utZapytanie.uiReadQuantity := 1;
		intOdczytCyklicznyTablica := intZnacznikDriveraOdczytuCyklicznego;
		intZnacznikOdczytuCyklicznegoReferencja := intZnacznikDriveraOdczytuCyklicznego;
		intZnacznikPomocniczy := intZnacznikDriveraOdczytuCyklicznego + 1;
		IF arOdczytCykliczny[intZnacznikPomocniczy].bAdresUrzadzenia = 0 THEN
			intZnacznikPomocniczy := 1;
		END_IF

// sprawdzenie czy następne żądanie nie jest w kolejności do bieżącego jeśli tak to grupuje je w jedno zapytanie

		WHILE (arOdczytCykliczny[intZnacznikPomocniczy].uiAdresRejestru - arOdczytCykliczny[intZnacznikDriveraOdczytuCyklicznego].uiAdresRejestru = 1 AND
				arOdczytCykliczny[intZnacznikPomocniczy].bFunkcja = arOdczytCykliczny[intZnacznikDriveraOdczytuCyklicznego].bFunkcja AND
				arOdczytCykliczny[intZnacznikPomocniczy].bAdresUrzadzenia = arOdczytCykliczny[intZnacznikDriveraOdczytuCyklicznego].bAdresUrzadzenia) DO
				
			utZapytanie.uiReadQuantity := utZapytanie.uiReadQuantity + 1;
			intZnacznikDriveraOdczytuCyklicznego := intZnacznikDriveraOdczytuCyklicznego + 1;
			IF arOdczytCykliczny[intZnacznikDriveraOdczytuCyklicznego].bAdresUrzadzenia = 0 THEN
				intZnacznikDriveraOdczytuCyklicznego := 1;
			END_IF
			intZnacznikPomocniczy := intZnacznikDriveraOdczytuCyklicznego + 1;
			IF arOdczytCykliczny[intZnacznikPomocniczy].bAdresUrzadzenia = 0 THEN
				intZnacznikPomocniczy := 1;
			END_IF
		END_WHILE
		intOdczytCyklicznyTablicaIlosc := UINT_TO_INT(utZapytanie.uiReadQuantity);
	END_IF
END_IF

// driver komunikacyjny MODBUS RTU

ModbusMasterRTU(xConnect := 		TRUE , 
				I_Port := 			arRTUParametryKomunikacji[utZapytanie.bUnitId].typNazwaPortuKomunikacyjnego , 
				eFrameType := 		arRTUParametryKomunikacji[utZapytanie.bUnitId].eTypRamki , 
				udiBaudrate := 		arRTUParametryKomunikacji[utZapytanie.bUnitId].udiPredkosc , 
				usiDataBits := 		arRTUParametryKomunikacji[utZapytanie.bUnitId].usiBityDanych , 
				eParity := 			arRTUParametryKomunikacji[utZapytanie.bUnitId].eParzystosc , 
				eStopBits := 		arRTUParametryKomunikacji[utZapytanie.bUnitId].eBityStopu , 
				eHandshake :=		arRTUParametryKomunikacji[utZapytanie.bUnitId].eHandshake , 
				ePhysical := 		arRTUParametryKomunikacji[utZapytanie.bUnitId].eDuplex , 
				tTimeOut := 		arRTUParametryKomunikacji[utZapytanie.bUnitId].tTimeout , 

				xTrigger := 		xDriverWykonajKomunikacje , 
				utQuery := 			utZapytanie , 
				utResponse := 		utOdpowiedz ,
 
				xError => 			xBladKomunikacji);

// obługa akcji po zakończeniu zadania komunikacji (zapis wartości , zapis błędu itd)
	
negWykonaj(CLK := xDriverWykonajKomunikacje);

IF negWykonaj.Q THEN
// jeżeli był błąd komunikacji wpisz go do tablicy błędów

	IF xBladKomunikacji THEN
		arStatusKomunikacji[utZapytanie.bUnitId] := enumModbusStatus.BrakKomunikacji;
		statusbledu := ModbusMasterRTU.oStatus;
		jakiezapytanie := utZapytanie;
		arStatusKomunikacjiTimestampOstatniBlad[utZapytanie.bUnitId] := _GetLongTime();
		IF utZapytaniePoprz.bFunctionCode = 0 THEN
			utZapytaniePoprz := utZapytanie;
		END_IF
		IF arRTUParametryKomunikacjiPoprz[3].udiPredkosc = 0 THEN
			arRTUParametryKomunikacjiPoprz := arRTUParametryKomunikacji;
		END_IF
	ELSE
		IF _GetLongTime() - arStatusKomunikacjiTimestampOstatniBlad[utZapytanie.bUnitId] > tCzasStabilnosciKomunikacji AND arStatusKomunikacji[utZapytanie.bUnitId] <> enumModbusStatus.KomunikacjaPrawidlowa THEN	
			arStatusKomunikacji[utZapytanie.bUnitId] := enumModbusStatus.KomunikacjaPrawidlowa;
		END_IF

// jeżeli zapytanie było żądaniem  wysłania danych

		IF utZapytanie.bFunctionCode = enumModbusKodyFunkcji.OdczytWejscBitowych OR utZapytanie.bFunctionCode = enumModbusKodyFunkcji.OdczytWyjscBitowych OR
			utZapytanie.bFunctionCode = enumModbusKodyFunkcji.OdczytNRejestrow OR utZapytanie.bFunctionCode = enumModbusKodyFunkcji.OdczytNRejestrowWejsciowych THEN
			intZnacznikOdczytuCyklicznegoPoczatek := 0;
		
// jeżeli był wykonany rozkaz odczytu danych z cyklu "na żądanie" - DOŁOŻONO KAWAŁEK KODU DEBUGUJĄCEGO - ZATRZYMYWANIE SIĘ STEROWNIKA NA ZAREMOWANEJ LINII

			IF intOdczytZadanieTablica <> 0 THEN
				arDebugZapytanie[intDebugZnacznik] := utZapytanie;
				arDebugOdpowiedz[intDebugZnacznik] := utOdpowiedz;
				typDebugOdczytZapisZadanie[intDebugZnacznik] := arOdczytZapisZadanie[intZnacznikDriveraOdczytuZapisuZadanie];				
				arDebugCzas[intDebugZnacznik] := FuGetDateAndTime();
				fnTablicaKomunikatowInkrementacja(intRozmiarTablicy := 900, intWskaznik := intDebugZnacznik);
//				arOdczytZapisZadanie[intZnacznikDriveraOdczytuZapisuZadanie].pZmiennaDoOdczytu^ := utOdpowiedz.awData[0];
			END_IF

// jeżeli był wykonany rozkaz odczytu danych z cyklu "cykliczny"

			IF intOdczytCyklicznyTablica <> 0 THEN
				intLoopOverflow:=1;
				FOR intLoop := 1 TO intOdczytCyklicznyTablicaIlosc DO
					IF arOdczytCykliczny[intOdczytCyklicznyTablica + intLoop - 1].pZmiennaReferencyjna <> null THEN
					arOdczytCykliczny[intOdczytCyklicznyTablica + intLoop - 1].pZmiennaReferencyjna^ := utOdpowiedz.awData[intLoop - 1];
					arOdczytCykliczny[intOdczytCyklicznyTablica + intLoop - 1].ltZnacznikCzasuWyslania := _GetLongTime();
					ELSE
					arOdczytCykliczny[intLoopOverflow].pZmiennaReferencyjna^ := utOdpowiedz.awData[intLoop - 1];
					arOdczytCykliczny[intLoopOverflow].ltZnacznikCzasuWyslania := _GetLongTime();
					intLoopOverflow:=intLoopOverflow+1;
					END_IF
				END_FOR
			END_IF
		END_IF
	END_IF
	intOdczytZadanieTablica := 0;
	intOdczytCyklicznyTablica := 0;
	intOdczytCyklicznyTablicaIlosc := 0;
END_IF


          
END_FUNCTION_BLOCK

FUNCTION_BLOCK fbModbusDriverTCP
  VAR_INPUT
    intOdczytZapisZadanieRozmiarBufora : INT;
    arTCPParametryKomunikacji : typModbusTCPParametryKomunikacji;
  END_VAR
  VAR_IN_OUT
    arOdczytCykliczny : ARRAY[1..1000] OF typModbusOdczytCykliczny;
    arOdczytZapisZadanie : ARRAY[1..1000] OF typModbusOdczytZapisZadanie;
    arStatusKomunikacji : ARRAY[1..256] OF INT;
    intZnacznikOdczytuZapisuZadanie : INT;
  END_VAR
  VAR
    ModbusMasterTCP : FbMbMasterTcp;
    utZapytanie : typMBQuery;
    utOdpowiedz : typMbResponse;
    xStatusPolaczenia : BOOL;
    xBladKomunikacji : BOOL;
    typStatusKomunikacji : WagoSysErrorBase.FbResult;
    fbTimerRestartuPolaczenia : TON;
    tCzasRestartuPolaczenia : TIME := TIME#15s0ms;
    tCzasPonowienia : LTIME := LTIME#15s0ms0us0ns;
    tCzasStabilnosciKomunikacji : LTIME := LTIME#30s0ms0us0ns;  (* czas po jakim driver raportuje poprawną komunikację po jej faktycznym odzyskaniu - czas powinien być większy niż czas tCzasPonawiania *)
    xDriverWykonajKomunikacje : BOOL;
    arStatusKomunikacjiTimestampOstatniaProba : ARRAY[1..256] OF LTIME;
    arStatusKomunikacjiTimestampOstatniBlad : ARRAY[1..256] OF LTIME;
    negWykonaj : F_TRIG;
    intZnacznikDriveraOdczytuCyklicznego : INT := 1;
    intZnacznikDriveraOdczytuZapisuZadanie : INT := 1;
    intZnacznikOdczytuCyklicznegoReferencja : INT;
    intZnacznikOdczytuCyklicznegoPoczatek : INT;
    intZnacznikOdczytuZapisuZadanieReferencja : INT;
    intZnacznikPomocniczy : INT;
    intOdczytZadanieTablica : INT;
    intOdczytCyklicznyTablica : INT;
    intOdczytCyklicznyTablicaIlosc : INT;
    intLoop : INT;
    intDebugZnacznik : INT;  (* debug *)
    arDebugZapytanie : ARRAY[0..1000] OF typMBQuery;
    arDebugOdpowiedz : ARRAY[0..1000] OF typMbResponse;
    typDebugOdczytZapisZadanie : ARRAY[0..1000] OF typModbusOdczytZapisZadanie;
    arDebugCzas : ARRAY[0..1000] OF DT;
  END_VAR

            // obsługa odczytu zapisu danych na żądanie

IF intZnacznikDriveraOdczytuZapisuZadanie <> intZnacznikOdczytuZapisuZadanie AND NOT xDriverWykonajKomunikacje THEN
	fnTablicaKomunikatowInkrementacja(intRozmiarTablicy := intOdczytZapisZadanieRozmiarBufora, intWskaznik := intZnacznikDriveraOdczytuZapisuZadanie);
	IF arStatusKomunikacji[arOdczytZapisZadanie[intZnacznikDriveraOdczytuZapisuZadanie].bAdresUrzadzenia] = enumModbusStatus.KomunikacjaPrawidlowa  AND xStatusPolaczenia THEN
		xDriverWykonajKomunikacje := TRUE;
		utZapytanie.bUnitId := arOdczytZapisZadanie[intZnacznikDriveraOdczytuZapisuZadanie].bAdresUrzadzenia;
		utZapytanie.bFunctionCode := arOdczytZapisZadanie[intZnacznikDriveraOdczytuZapisuZadanie].bFunkcja;
		utZapytanie.uiReadQuantity := 1;
		utZapytanie.uiReadAddress := arOdczytZapisZadanie[intZnacznikDriveraOdczytuZapisuZadanie].uiAdresRejestru;
		utZapytanie.uiWriteAddress := arOdczytZapisZadanie[intZnacznikDriveraOdczytuZapisuZadanie].uiAdresRejestru;
		utZapytanie.awWriteData[0] := arOdczytZapisZadanie[intZnacznikDriveraOdczytuZapisuZadanie].wWartoscDoZapisania;
		utZapytanie.uiWriteQuantity := 1;
		intOdczytZadanieTablica := intZnacznikDriveraOdczytuZapisuZadanie;
	END_IF
END_IF

// obsługa odczytu zmiennych zapisanych w tabeli

IF NOT xDriverWykonajKomunikacje AND xStatusPolaczenia AND NOT xBladKomunikacji THEN

	intZnacznikOdczytuCyklicznegoReferencja := intZnacznikDriveraOdczytuCyklicznego;
	intZnacznikDriveraOdczytuCyklicznego := intZnacznikDriveraOdczytuCyklicznego + 1;
	IF arOdczytCykliczny[intZnacznikDriveraOdczytuCyklicznego].bAdresUrzadzenia = 0 THEN
		intZnacznikDriveraOdczytuCyklicznego := 1;
	END_IF

	WHILE intZnacznikOdczytuCyklicznegoReferencja <> intZnacznikDriveraOdczytuCyklicznego AND _GetLongTime() - arStatusKomunikacjiTimestampOstatniaProba[arOdczytCykliczny[intZnacznikDriveraOdczytuCyklicznego].bAdresUrzadzenia] < tCzasPonowienia AND
			_GetLongTime() - arOdczytCykliczny[intZnacznikDriveraOdczytuCyklicznego].ltZnacznikCzasuWyslania < arOdczytCykliczny[intZnacznikDriveraOdczytuCyklicznego].ltCzestotliwosc DO
		intZnacznikDriveraOdczytuCyklicznego := intZnacznikDriveraOdczytuCyklicznego + 1;
		IF arOdczytCykliczny[intZnacznikDriveraOdczytuCyklicznego].bAdresUrzadzenia = 0 THEN
			intZnacznikDriveraOdczytuCyklicznego := 1;
		END_IF
	END_WHILE

// zapis adresu startowego rejestrów do zapisu

	IF intZnacznikOdczytuCyklicznegoReferencja <> intZnacznikDriveraOdczytuCyklicznego THEN
		xDriverWykonajKomunikacje := TRUE;
		arStatusKomunikacjiTimestampOstatniaProba[arOdczytCykliczny[intZnacznikDriveraOdczytuCyklicznego].bAdresUrzadzenia] := _GetLongTime();
		utZapytanie.bUnitId := arOdczytCykliczny[intZnacznikDriveraOdczytuCyklicznego].bAdresUrzadzenia;
		utZapytanie.bFunctionCode := arOdczytCykliczny[intZnacznikDriveraOdczytuCyklicznego].bFunkcja;
		utZapytanie.uiReadAddress := arOdczytCykliczny[intZnacznikDriveraOdczytuCyklicznego].uiAdresRejestru;
		utZapytanie.uiReadQuantity := 1;
		intOdczytCyklicznyTablica := intZnacznikDriveraOdczytuCyklicznego;
		intZnacznikOdczytuCyklicznegoReferencja := intZnacznikDriveraOdczytuCyklicznego;
		intZnacznikPomocniczy := intZnacznikDriveraOdczytuCyklicznego + 1;
		IF arOdczytCykliczny[intZnacznikPomocniczy].bAdresUrzadzenia = 0 THEN
			intZnacznikPomocniczy := 1;
		END_IF

// sprawdzenie czy następne żądanie nie jest w kolejności do bieżącego jeśli tak to grupuje je w jedno zapytanie

		WHILE (arOdczytCykliczny[intZnacznikPomocniczy].uiAdresRejestru - arOdczytCykliczny[intZnacznikDriveraOdczytuCyklicznego].uiAdresRejestru = 1 AND
				arOdczytCykliczny[intZnacznikPomocniczy].bFunkcja = arOdczytCykliczny[intZnacznikDriveraOdczytuCyklicznego].bFunkcja AND
				arOdczytCykliczny[intZnacznikPomocniczy].bAdresUrzadzenia = arOdczytCykliczny[intZnacznikDriveraOdczytuCyklicznego].bAdresUrzadzenia) DO
				
			utZapytanie.uiReadQuantity := utZapytanie.uiReadQuantity + 1;
			intZnacznikDriveraOdczytuCyklicznego := intZnacznikDriveraOdczytuCyklicznego + 1;
			IF arOdczytCykliczny[intZnacznikDriveraOdczytuCyklicznego].bAdresUrzadzenia = 0 THEN
				intZnacznikDriveraOdczytuCyklicznego := 1;
			END_IF
			intZnacznikPomocniczy := intZnacznikDriveraOdczytuCyklicznego + 1;
			IF arOdczytCykliczny[intZnacznikPomocniczy].bAdresUrzadzenia = 0 THEN
				intZnacznikPomocniczy := 1;
			END_IF
		END_WHILE
		intOdczytCyklicznyTablicaIlosc := UINT_TO_INT(utZapytanie.uiReadQuantity);
	END_IF
END_IF

// restart połączenia jeśli brak komunikacji

fbTimerRestartuPolaczenia(IN := (NOT xStatusPolaczenia OR xBladKomunikacji) AND NOT fbTimerRestartuPolaczenia.Q, PT := tCzasRestartuPolaczenia);

// driver komunikacyjny MODBUS TCP

ModbusMasterTCP(xConnect :=			NOT fbTimerRestartuPolaczenia.Q ,
				sHost :=			arTCPParametryKomunikacji.sAdresTCP ,
				wPort := 			arTCPParametryKomunikacji.wPortTCP ,
				utKeepAlive := 		arTCPParametryKomunikacji.utPodtrzymajWtyczkeTCP ,
				eFrameType := 		arTCPParametryKomunikacji.eTypRamki ,
				tTimeOut := 		arTCPParametryKomunikacji.tTimeOut ,
					
				xIsOpen => 			xStatusPolaczenia ,
				xError => 			xBladKomunikacji ,
				oStatus => 			typStatusKomunikacji ,
					
				xTrigger := 		xDriverWykonajKomunikacje , 
				utQuery := 			utZapytanie , 
				utResponse := 		utOdpowiedz);

// obługa akcji po zakończeniu zadania komunikacji (zapis wartości , zapis błędu itd)
	
negWykonaj(CLK := xDriverWykonajKomunikacje);

IF negWykonaj.Q THEN
// jeżeli był błąd komunikacji wpisz go do tablicy błędów

	IF xBladKomunikacji THEN
		arStatusKomunikacji[utZapytanie.bUnitId] := enumModbusStatus.BrakKomunikacji;
		arStatusKomunikacjiTimestampOstatniBlad[utZapytanie.bUnitId] := _GetLongTime();
		ELSE
		IF _GetLongTime() - arStatusKomunikacjiTimestampOstatniBlad[utZapytanie.bUnitId] > tCzasStabilnosciKomunikacji AND arStatusKomunikacji[utZapytanie.bUnitId] <> enumModbusStatus.KomunikacjaPrawidlowa THEN	
			arStatusKomunikacji[utZapytanie.bUnitId] := enumModbusStatus.KomunikacjaPrawidlowa;
		END_IF

// jeżeli zapytanie było żądaniem  wysłania danych

		IF utZapytanie.bFunctionCode = enumModbusKodyFunkcji.OdczytWejscBitowych OR utZapytanie.bFunctionCode = enumModbusKodyFunkcji.OdczytWyjscBitowych OR
			utZapytanie.bFunctionCode = enumModbusKodyFunkcji.OdczytNRejestrow OR utZapytanie.bFunctionCode = enumModbusKodyFunkcji.OdczytNRejestrowWejsciowych THEN
			intZnacznikOdczytuCyklicznegoPoczatek := 0;
		
// jeżeli był wykonany rozkaz odczytu danych z cyklu "na żądanie"

			IF intOdczytZadanieTablica <> 0 THEN
				arDebugZapytanie[intDebugZnacznik] := utZapytanie;
				arDebugOdpowiedz[intDebugZnacznik] := utOdpowiedz;
				typDebugOdczytZapisZadanie[intDebugZnacznik] := arOdczytZapisZadanie[intZnacznikDriveraOdczytuZapisuZadanie];				
				arDebugCzas[intDebugZnacznik] := FuGetDateAndTime();
				fnTablicaKomunikatowInkrementacja(intRozmiarTablicy := 900, intWskaznik := intDebugZnacznik);
//				arOdczytZapisZadanie[intZnacznikDriveraOdczytuZapisuZadanie].pZmiennaDoOdczytu^ := utOdpowiedz.awData[0];
			END_IF

// jeżeli był wykonany rozkaz odczytu danych z cyklu "cykliczny"

			IF intOdczytCyklicznyTablica <> 0 THEN
				FOR intLoop := 1 TO intOdczytCyklicznyTablicaIlosc DO
					arOdczytCykliczny[intOdczytCyklicznyTablica + intLoop - 1].pZmiennaReferencyjna^ := utOdpowiedz.awData[intLoop - 1];
					arOdczytCykliczny[intOdczytCyklicznyTablica + intLoop - 1].ltZnacznikCzasuWyslania := _GetLongTime();
				END_FOR
			END_IF
		END_IF
	END_IF
	intOdczytZadanieTablica := 0;
	intOdczytCyklicznyTablica := 0;
	intOdczytCyklicznyTablicaIlosc := 0;
END_IF
          
END_FUNCTION_BLOCK

FUNCTION_BLOCK fbModbusOdczytZapis
  VAR_INPUT
    intModbusOdczytZapisZadanieRozmiar : INT;  (* Rozmiar tablicy danych modbusa *)
    xOdczytajRejestr : BOOL;  (* Żądanie odczytania rejestru *)
    bAdresOdczyt : BYTE := 2#101000;  (* Adres urządzenia, z którego ma zostać dokonany odczyt *)
    uiAdresRejestruOdczyt : UINT := 2010;  (* Adres rejestru, z którego ma zostać dokonany odczyt *)
    xZapiszRejestr : BOOL;  (* Żądanie zapisania rejestru *)
    bAdresZapis : BYTE;  (* Adres urządzenia, na który ma zostać dokonany zapis *)
    uiAdresRejestruZapis : UINT;  (* Adres rejestru, na który ma zostać dokonany zapis *)
    wZawartoscRejestruZapis : WORD;  (* Dane do zapisu *)
  END_VAR
  VAR_IN_OUT
    arModbusOdczytCykliczny : ARRAY[1..5000] OF typModbusOdczytCykliczny;
    arModbusOdczytZapisZadanie : ARRAY[1..1000] OF typModbusOdczytZapisZadanie;
    intModbusOdczytZapisZadanieZnacznikZapisu : INT;
  END_VAR
  VAR
    tMinimalnyCzasRaportowania : TIME := TIME#15s0ms;
    intPetlaPierwszySkan : INT := 1;
    wZawartoscRejestruOdczyt : WORD;  (* Zawartość odczytanego rejestru *)
    xPierwszyCykl : BOOL := TRUE;  (* Pierwszy cykl programu *)
  END_VAR

            (*			
Autor:					Artur Wyszomirski, 2019-10-11 
Prawa majątkowe: 		Solwena Sp. z o.o., 
Aktualizacje:			2019-10-22: - dodanie wyszukiwania wolnego miejsca w tablicy arModbusOdczytCykliczny
									- wprowadzenie domyślnych wartości dla bAdresOdczyt i uiAdresRejestruOdczyt
									- przypisywanie wartości ltCzestotliwosc i pZmiennaReferencyjna w pierwszym cyklu programu

Opis:					Odczyt i zapis dowolnego rejestru Modbus				
*)

// Pierwszy cykl programu
IF xPierwszyCykl THEN
	WHILE arModbusOdczytCykliczny[intPetlaPierwszySkan].bAdresUrzadzenia <> 0 DO
		intPetlaPierwszySkan := intPetlaPierwszySkan + 1;
	END_WHILE
END_IF

// Odczyt
IF xPierwszyCykl THEN
	arModbusOdczytCykliczny[intPetlaPierwszySkan].ltCzestotliwosc := TIME_TO_LTIME(tMinimalnyCzasRaportowania);
	arModbusOdczytCykliczny[intPetlaPierwszySkan].pZmiennaReferencyjna := ADR(wZawartoscRejestruOdczyt);
END_IF
IF xOdczytajRejestr OR xPierwszyCykl THEN
	arModbusOdczytCykliczny[intPetlaPierwszySkan].bAdresUrzadzenia := bAdresOdczyt;
	arModbusOdczytCykliczny[intPetlaPierwszySkan].bFunkcja := TO_BYTE(enumModbusKodyFunkcji.OdczytNRejestrow);
	arModbusOdczytCykliczny[intPetlaPierwszySkan].uiAdresRejestru := uiAdresRejestruOdczyt;

END_IF

// Zapis
IF xZapiszRejestr THEN
	fnModbusZapisRejestru(	bAdresUrzadzenia := bAdresZapis,
							bFunkcja := INT_TO_BYTE(enumModbusKodyFunkcji.ZapisRejestru),
							uiAdresRejestru := uiAdresRejestruZapis,
							pZmiennaReferencyjna := 0,
							wWartoscDoZapisania := wZawartoscRejestruZapis,
							intModbusOdczytZapisZadanieRozmiar := intModbusOdczytZapisZadanieRozmiar,
							arModbusOdczytZapisZadanie := arModbusOdczytZapisZadanie,
							intModbusOdczytZapisZadanieZnacznikZapisu := intModbusOdczytZapisZadanieZnacznikZapisu);
END_IF
	
xPierwszyCykl := FALSE;
          
END_FUNCTION_BLOCK

FUNCTION_BLOCK fbPPPSAnalizatorDirisA40
  VAR_INPUT
    sKomunikat : alSTRINGKomunikat;  (* komunikat z systemu zewnętrznego *)
    intTablicaKomunikatowRozmiar : INT;  (* rozmiar tablicy danych wysyłkowych *)
    xTablicaKomunikatowHold : BOOL;  (* wstrzymanie komunikacji mniej ważnych komunikatów *)
    sIdInstancji : STRING;  (* parametr ID rolety np NS02L*202IBM**** *)
    sIdAplikacji : STRING;  (* parametr ID aplikacji np SO*******ECL*000 *)
    sMnemonik : STRING;  (* mnemonik właściciela - BCB* *)
    sMACAdres : STRING;  (* MAC adres sterownika *)
    sDaneZapasowe : STRING;  (* 6 znaków zapasu *)
    tCzasOpoznieniaRestartu : TIME;  (* czas opóźnienia po którym zaczynają być raportowane wartości *)
    bAdres : BYTE;
    rDeadband : REAL;
    tMinimalnyCzasRaportowania : TIME;
    tMaksymalnyCzasRaportowania : TIME;
    xAutonomizacja : BOOL;
  END_VAR
  VAR_IN_OUT
    arModbusOdczytCykliczny : ARRAY[1..5000] OF typModbusOdczytCykliczny;
    arModbusStatusKomunikacji : ARRAY[1..256] OF INT;
    arTablicaKomunikatow : alARRAYTablicaKomunikatow;
    intTablicaKomunikatowZnacznikZapisu : INT;
  END_VAR
  VAR
    xPierwszySkan : BOOL := TRUE;
    intPetlaPierwszySkan : INT := 1;
    fbTimerBrakuKomunikacji : TON;  (* Kontrola komunikacji urządzenia *)
    xBrakKomunikacjiPLC : BOOL;
    xBrakKomunikacjiIZE : BOOL;
    wNapiecieL1Hi : WORD;  (* Napięcia fazowe *)
    wNapiecieL1Lo : WORD;
    rNapiecieL1 : REAL;
    fbNapiecieL1 : fbFiltrWartoscAnalogowa;
    rNapiecieL1Zaraportowana : REAL;
    rNapiecieL1Pamiec : REAL;
    xBrakZmianyNapiecieL1 : BOOL;
    fbBrakZmianyNapiecieL1Timer : TON;
    xBladBrakZmianyNapiecieL1 : BOOL;
    wNapiecieL2Hi : WORD;
    wNapiecieL2Lo : WORD;
    rNapiecieL2 : REAL;
    fbNapiecieL2 : fbFiltrWartoscAnalogowa;
    rNapiecieL2Zaraportowana : REAL;
    rNapiecieL2Pamiec : REAL;
    xBrakZmianyNapiecieL2 : BOOL;
    fbBrakZmianyNapiecieL2Timer : TON;
    xBladBrakZmianyNapiecieL2 : BOOL;
    wNapiecieL3Hi : WORD;
    wNapiecieL3Lo : WORD;
    rNapiecieL3 : REAL;
    fbNapiecieL3 : fbFiltrWartoscAnalogowa;
    rNapiecieL3Zaraportowana : REAL;
    rNapiecieL3Pamiec : REAL;
    xBrakZmianyNapiecieL3 : BOOL;
    fbBrakZmianyNapiecieL3Timer : TON;
    xBladBrakZmianyNapiecieL3 : BOOL;
    wNapiecieL1L2Hi : WORD;  (* Napięcia przewodowe *)
    wNapiecieL1L2Lo : WORD;
    rNapiecieL1L2 : REAL;
    fbNapiecieL1L2 : fbFiltrWartoscAnalogowa;
    rNapiecieL1L2Zaraportowana : REAL;
    wNapiecieL2L3Hi : WORD;
    wNapiecieL2L3Lo : WORD;
    rNapiecieL2L3 : REAL;
    fbNapiecieL2L3 : fbFiltrWartoscAnalogowa;
    rNapiecieL2L3Zaraportowana : REAL;
    wNapiecieL3L1Hi : WORD;
    wNapiecieL3L1Lo : WORD;
    rNapiecieL3L1 : REAL;
    fbNapiecieL3L1 : fbFiltrWartoscAnalogowa;
    rNapiecieL3L1Zaraportowana : REAL;
    wCzestotliwoscHi : WORD;  (* Częstotliwość *)
    wCzestotliwoscLo : WORD;
    rCzestotliwosc : REAL;
    fbCzestotliwosc : fbFiltrWartoscAnalogowa;
    rCzestotliwoscZaraportowana : REAL;
    wCzasPracyAnalizatoraHi : WORD;  (* Czas pracy *)
    wCzasPracyAnalizatoraLo : WORD;
    rCzasPracyAnalizatora : REAL;
    fbCzasPracyAnalizatora : fbFiltrWartoscAnalogowa;
    rCzasPracyAnalizatoraZaraportowana : REAL;
    wPradL1Hi : WORD;  (* Prądy fazowe *)
    wPradL1Lo : WORD;
    rPradL1 : REAL;
    fbPradL1 : fbFiltrWartoscAnalogowa;
    rPradL1Zaraportowana : REAL;
    rPradL1Pamiec : REAL;
    xBrakZmianyPradL1 : BOOL;
    fbBrakZmianyPradL1Timer : TON;
    xBladBrakZmianyPradL1 : BOOL;
    wPradL2Hi : WORD;
    wPradL2Lo : WORD;
    rPradL2 : REAL;
    fbPradL2 : fbFiltrWartoscAnalogowa;
    rPradL2Zaraportowana : REAL;
    rPradL2Pamiec : REAL;
    xBrakZmianyPradL2 : BOOL;
    fbBrakZmianyPradL2Timer : TON;
    xBladBrakZmianyPradL2 : BOOL;
    wPradL3Hi : WORD;
    wPradL3Lo : WORD;
    rPradL3 : REAL;
    fbPradL3 : fbFiltrWartoscAnalogowa;
    rPradL3Zaraportowana : REAL;
    rPradL3Pamiec : REAL;
    xBrakZmianyPradL3 : BOOL;
    fbBrakZmianyPradL3Timer : TON;
    xBladBrakZmianyPradL3 : BOOL;
    wPradNHi : WORD;
    wPradNLo : WORD;
    rPradN : REAL;
    fbPradN : fbFiltrWartoscAnalogowa;
    rPradNZaraportowana : REAL;
    wPradSredniL1Hi : WORD;  (* Prądy średnie fazowe *)
    wPradSredniL1Lo : WORD;
    rPradSredniL1 : REAL;
    fbPradSredniL1 : fbFiltrWartoscAnalogowa;
    rPradSredniL1Zaraportowana : REAL;
    wPradSredniL2Hi : WORD;
    wPradSredniL2Lo : WORD;
    rPradSredniL2 : REAL;
    fbPradSredniL2 : fbFiltrWartoscAnalogowa;
    rPradSredniL2Zaraportowana : REAL;
    wPradSredniL3Hi : WORD;
    wPradSredniL3Lo : WORD;
    rPradSredniL3 : REAL;
    fbPradSredniL3 : fbFiltrWartoscAnalogowa;
    rPradSredniL3Zaraportowana : REAL;
    rPradSredni : REAL;  (* Prąd średni (I1+I2+I3)/3 *)
    fbPradSredni : fbFiltrWartoscAnalogowa;
    rPradSredniZaraportowana : REAL;
    wMocCzynnaCalkowitaHi : WORD;  (* Moc 3-fazowa czynna *)
    wMocCzynnaCalkowitaLo : WORD;
    rMocCzynnaCalkowita : REAL;
    fbMocCzynnaCalkowita : fbFiltrWartoscAnalogowa;
    rMocCzynnaCalkowitaZaraportowana : REAL;
    wMocBiernaCalkowitaHi : WORD;  (* Moc 3-fazowa bierna *)
    wMocBiernaCalkowitaLo : WORD;
    rMocBiernaCalkowita : REAL;
    fbMocBiernaCalkowita : fbFiltrWartoscAnalogowa;
    rMocBiernaCalkowitaZaraportowana : REAL;
    wMocPozornaCalkowitaHi : WORD;  (* Moc 3-fazowa pozorna *)
    wMocPozornaCalkowitaLo : WORD;
    rMocPozornaCalkowita : REAL;
    fbMocPozornaCalkowita : fbFiltrWartoscAnalogowa;
    rMocPozornaCalkowitaZaraportowana : REAL;
    wWspolczynnikMocyCalkowityHi : WORD;  (* Całkowity współczynnik mocy *)
    wWspolczynnikMocyCalkowityLo : WORD;
    rWspolczynnikMocyCalkowity : REAL;
    fbWspolczynnikMocyCalkowity : fbFiltrWartoscAnalogowa;
    rWspolczynnikMocyCalkowityZaraportowana : REAL;
    wMocCzynnaL1Hi : WORD;  (* Moc Czynna fazowa *)
    wMocCzynnaL1Lo : WORD;
    rMocCzynnaL1 : REAL;
    fbMocCzynnaL1 : fbFiltrWartoscAnalogowa;
    rMocCzynnaL1Zaraportowana : REAL;
    wMocCzynnaL2Hi : WORD;
    wMocCzynnaL2Lo : WORD;
    rMocCzynnaL2 : REAL;
    fbMocCzynnaL2 : fbFiltrWartoscAnalogowa;
    rMocCzynnaL2Zaraportowana : REAL;
    wMocCzynnaL3Hi : WORD;
    wMocCzynnaL3Lo : WORD;
    rMocCzynnaL3 : REAL;
    fbMocCzynnaL3 : fbFiltrWartoscAnalogowa;
    rMocCzynnaL3Zaraportowana : REAL;
    wMocBiernaL1Hi : WORD;  (* Moc Bierna fazowa *)
    wMocBiernaL1Lo : WORD;
    rMocBiernaL1 : REAL;
    fbMocBiernaL1 : fbFiltrWartoscAnalogowa;
    rMocBiernaL1Zaraportowana : REAL;
    wMocBiernaL2Hi : WORD;
    wMocBiernaL2Lo : WORD;
    rMocBiernaL2 : REAL;
    fbMocBiernaL2 : fbFiltrWartoscAnalogowa;
    rMocBiernaL2Zaraportowana : REAL;
    wMocBiernaL3Hi : WORD;
    wMocBiernaL3Lo : WORD;
    rMocBiernaL3 : REAL;
    fbMocBiernaL3 : fbFiltrWartoscAnalogowa;
    rMocBiernaL3Zaraportowana : REAL;
    wMocPozornaL1Hi : WORD;  (* Moc Pozorna fazowa *)
    wMocPozornaL1Lo : WORD;
    rMocPozornaL1 : REAL;
    fbMocPozornaL1 : fbFiltrWartoscAnalogowa;
    rMocPozornaL1Zaraportowana : REAL;
    wMocPozornaL2Hi : WORD;
    wMocPozornaL2Lo : WORD;
    rMocPozornaL2 : REAL;
    fbMocPozornaL2 : fbFiltrWartoscAnalogowa;
    rMocPozornaL2Zaraportowana : REAL;
    wMocPozornaL3Hi : WORD;
    wMocPozornaL3Lo : WORD;
    rMocPozornaL3 : REAL;
    fbMocPozornaL3 : fbFiltrWartoscAnalogowa;
    rMocPozornaL3Zaraportowana : REAL;
    wWspolczynnikMocyL1Hi : WORD;  (* Fazowe współczynniki mocy *)
    wWspolczynnikMocyL1Lo : WORD;
    rWspolczynnikMocyL1 : REAL;
    fbWspolczynnikMocyL1 : fbFiltrWartoscAnalogowa;
    rWspolczynnikMocyL1Zaraportowana : REAL;
    wWspolczynnikMocyL2Hi : WORD;
    wWspolczynnikMocyL2Lo : WORD;
    rWspolczynnikMocyL2 : REAL;
    fbWspolczynnikMocyL2 : fbFiltrWartoscAnalogowa;
    rWspolczynnikMocyL2Zaraportowana : REAL;
    wWspolczynnikMocyL3Hi : WORD;
    wWspolczynnikMocyL3Lo : WORD;
    rWspolczynnikMocyL3 : REAL;
    fbWspolczynnikMocyL3 : fbFiltrWartoscAnalogowa;
    rWspolczynnikMocyL3Zaraportowana : REAL;
    wEnergiaCzynnaPobranaHi : WORD;  (* Energia pobrana *)
    wEnergiaCzynnaPobranaLo : WORD;
    rEnergiaCzynnaPobrana : REAL;
    fbEnergiaCzynnaPobrana : fbFiltrWartoscAnalogowa;
    rEnergiaCzynnaPobranaZaraportowana : REAL;
    wEnergiaBiernaPobranaHi : WORD;
    wEnergiaBiernaPobranaLo : WORD;
    rEnergiaBiernaPobrana : REAL;
    fbEnergiaBiernaPobrana : fbFiltrWartoscAnalogowa;
    rEnergiaBiernaPobranaZaraportowana : REAL;
    wEnergiaPozornaPobranaHi : WORD;
    wEnergiaPozornaPobranaLo : WORD;
    rEnergiaPozornaPobrana : REAL;
    fbEnergiaPozornaPobrana : fbFiltrWartoscAnalogowa;
    rEnergiaPozornaPobranaZaraportowana : REAL;
    wMocCzynnaSredniaHi : WORD;  (* Moc średnia *)
    wMocCzynnaSredniaLo : WORD;
    rMocCzynnaSrednia : REAL;
    fbMocCzynnaSrednia : fbFiltrWartoscAnalogowa;
    rMocCzynnaSredniaZaraportowana : REAL;
    wMocBiernaSredniaHi : WORD;
    wMocBiernaSredniaLo : WORD;
    rMocBiernaSrednia : REAL;
    fbMocBiernaSrednia : fbFiltrWartoscAnalogowa;
    rMocBiernaSredniaZaraportowana : REAL;
    wMocPozornaSredniaHi : WORD;
    wMocPozornaSredniaLo : WORD;
    rMocPozornaSrednia : REAL;
    fbMocPozornaSrednia : fbFiltrWartoscAnalogowa;
    rMocPozornaSredniaZaraportowana : REAL;
    wMaksymalneNapiecieL1Hi : WORD;  (* Maksymalne napięcia fazowe *)
    wMaksymalneNapiecieL1Lo : WORD;
    rMaksymalneNapiecieL1 : REAL;
    fbMaksymalneNapiecieL1 : fbFiltrWartoscAnalogowa;
    rMaksymalneNapiecieL1Zaraportowana : REAL;
    wMaksymalneNapiecieL2Hi : WORD;
    wMaksymalneNapiecieL2Lo : WORD;
    rMaksymalneNapiecieL2 : REAL;
    fbMaksymalneNapiecieL2 : fbFiltrWartoscAnalogowa;
    rMaksymalneNapiecieL2Zaraportowana : REAL;
    wMaksymalneNapiecieL3Hi : WORD;
    wMaksymalneNapiecieL3Lo : WORD;
    rMaksymalneNapiecieL3 : REAL;
    fbMaksymalneNapiecieL3 : fbFiltrWartoscAnalogowa;
    rMaksymalneNapiecieL3Zaraportowana : REAL;
    wTHDNapieciaL1 : WORD;  (* THD napięcia *)
    rTHDNapieciaL1 : REAL;
    fbTHDNapieciaL1 : fbFiltrWartoscAnalogowa;
    rTHDNapieciaL1Zaraportowana : REAL;
    wTHDNapieciaL2 : WORD;
    rTHDNapieciaL2 : REAL;
    fbTHDNapieciaL2 : fbFiltrWartoscAnalogowa;
    rTHDNapieciaL2Zaraportowana : REAL;
    wTHDNapieciaL3 : WORD;
    rTHDNapieciaL3 : REAL;
    fbTHDNapieciaL3 : fbFiltrWartoscAnalogowa;
    rTHDNapieciaL3Zaraportowana : REAL;
    wTHDPraduL1 : WORD;  (* THD prądu *)
    rTHDPraduL1 : REAL;
    fbTHDPraduL1 : fbFiltrWartoscAnalogowa;
    rTHDPraduL1Zaraportowana : REAL;
    wTHDPraduL2 : WORD;
    rTHDPraduL2 : REAL;
    fbTHDPraduL2 : fbFiltrWartoscAnalogowa;
    rTHDPraduL2Zaraportowana : REAL;
    wTHDPraduL3 : WORD;
    rTHDPraduL3 : REAL;
    fbTHDPraduL3 : fbFiltrWartoscAnalogowa;
    rTHDPraduL3Zaraportowana : REAL;
    xPoInicjalizacji : BOOL;  (* inicjalizacja *)
    fbInicjalizacyjnyTimer : TON;
    intStatus : INT := enumPPPSUrzadenieStatus.Prawidlowy;  (* status urządzenia *)
    intStatusZaraportowana : INT;  (* status urządzenia zaraportowany *)
    sDane : alSTRINGKomunikat;
    sWyslanyKomunikat : alSTRINGKomunikat;
    xZadanieRaportu : BOOL;
    sWyslanyKomunikatDummy : alSTRINGKomunikat;
    sKomunikatPamiec : alSTRINGKomunikat;
    intPetla : INT;
    arErrorStan : ARRAY[0..20] OF INT;  (* tablica przechowująca statusy alarmowe *)
    arErrorKlasa : ARRAY[0..20] OF INT;  (* tablica przechowująca klasy danych alarmów *)
    xRaport : BOOL := FALSE;
    xOverFlow : BOOL;
  END_VAR

            (*			
Autor:					Paweł Kąkol, 2018-09-04-PK
Prawa majątkowe: 		Solwena Sp. z o.o., 
Opis:					fb służy do komunikacji po Modbus RTU z analizatorem sieci ECA0 na budynkach PPP Sopot
						Analizator Diris A40
						
Aktualizacje:			2018-11-20-JB: Poprawienie adresów Modbusowych
						2019-01-21-JC: Przeliczanie charakteru mocy biernej oraz współczynnika mocy (czynna/indukcyjna)
						2019-03-26-AWy: Wyłączenie (wykomentowanie) eneregii oddanej czynnej i biernej
						2019-04-01-AWy: Przeliczenie pomocnicze dla mocy czynnej całkowitej
						2019-05-05-AWy: Dodanie bloków włączania autonomizacji i kontroli komunikacji (analogicznie do pozostałych fb). Usunięcie zmiennej xBrakKomunikacji
						2019-08-14-AWy: Przeniesienie xAutonomizacja do VAR_INPUT
						2019-09-04-AWy: Usunięcie bugów z obliczania współczynnika mocy i mocy biernej.
						2019-09-05-Awy: Zmiana sposobu przeliczania wartości odczytanych po modbusie (sklejenie w DINT i konwersja na REAL). Usunięcie energii oddanej czynnej i biernej.
										Zmiana nazwy atrybutu FACTOR na FACTOR3PH.
						2019-10-18-JB: Zmiana dead-bandów.
						2019-10-24-AWy: Zmiana wartości tCzasMinimalny dla czasu pracy analizatora.
	
*)

//inicjalizacja sterownika

fbInicjalizacyjnyTimer(IN := NOT xPoInicjalizacji , PT := tCzasOpoznieniaRestartu);
IF fbInicjalizacyjnyTimer.Q THEN
	rNapiecieL1Zaraportowana := rNapiecieL1;
	rNapiecieL2Zaraportowana := rNapiecieL2;
	rNapiecieL3Zaraportowana :=sdfsdgsdf rNapiecieL3;
	rNapiecieL1L2Zaraportowana := rNapiecieL1L2;
	rNapiecieL2L3Zaraportowana := rNapiecieL2L3;
	rNapiecieL3L1Zaraportowana := rNapiecieL3L1;
	rCzestotliwoscZaraportowana := rCzestotliwosc;
	rCzasPracyAnalizatoraZaraportowana := rCzasPracyAnalizatora;
	rPradL1Zaraportowana := rPradL1;
	rPradL2Zaraportowana := rPradL2;
	rPradL3Zaraportowana := rPradL3;
	rPradNZaraportowana := rPradN;
	rPradSredniL1Zaraportowana := rPradSredniL1;
	rPradSredniL2Zaraportowana := rPradSredniL2;
	rPradSredniL3Zaraportowana := rPradSredniL3;
	rPradSredniZaraportowana := rPradSredni;
	rMocCzynnaCalkowitaZaraportowana := rMocCzynnaCalkowita;
	rMocBiernaCalkowitaZaraportowana := rMocBiernaCalkowita;
	rMocPozornaCalkowitaZaraportowana := rMocPozornaCalkowita;
	rWspolczynnikMocyCalkowityZaraportowana := rWspolczynnikMocyCalkowity;
	rMocCzynnaL1Zaraportowana := rMocCzynnaL1;
	rMocCzynnaL2Zaraportowana := rMocCzynnaL2;
	rMocCzynnaL3Zaraportowana := rMocCzynnaL3;
	rMocBiernaL1Zaraportowana := rMocBiernaL1;
	rMocBiernaL2Zaraportowana := rMocBiernaL2;
	rMocBiernaL3Zaraportowana := rMocBiernaL3;
	rMocPozornaL1Zaraportowana := rMocPozornaL1;
	rMocPozornaL2Zaraportowana := rMocPozornaL2;
	rMocPozornaL3Zaraportowana := rMocPozornaL3;
	rWspolczynnikMocyL1Zaraportowana := rWspolczynnikMocyL1;
	rWspolczynnikMocyL2Zaraportowana := rWspolczynnikMocyL2;
	rWspolczynnikMocyL3Zaraportowana := rWspolczynnikMocyL3;
	rEnergiaCzynnaPobranaZaraportowana := rEnergiaCzynnaPobrana;
	rEnergiaBiernaPobranaZaraportowana := rEnergiaBiernaPobrana;
	rEnergiaPozornaPobranaZaraportowana := rEnergiaPozornaPobrana;
	rMocCzynnaSredniaZaraportowana := rMocCzynnaSrednia;
	rMocBiernaSredniaZaraportowana := rMocBiernaSrednia;
	rMocPozornaSredniaZaraportowana := rMocPozornaSrednia;
	rMaksymalneNapiecieL1Zaraportowana := rMaksymalneNapiecieL1;
	rMaksymalneNapiecieL2Zaraportowana := rMaksymalneNapiecieL2;
	rMaksymalneNapiecieL3Zaraportowana := rMaksymalneNapiecieL3;
	rTHDNapieciaL1Zaraportowana := rTHDNapieciaL1;
	rTHDNapieciaL2Zaraportowana := rTHDNapieciaL2;
	rTHDNapieciaL3Zaraportowana := rTHDNapieciaL3;
	rTHDPraduL1Zaraportowana := rTHDPraduL1;
	rTHDPraduL2Zaraportowana := rTHDPraduL2;
	rTHDPraduL3Zaraportowana := rTHDPraduL3;
	intStatusZaraportowana := intStatus;
	xPoInicjalizacji := TRUE;
	dupa dupa dupa
END_IF

// Włącz autonomizację jeśli sterownik jest w stanie inicjalizacji lub nastąpiło wymuszenie autonomizacji
IF NOT xPoInicjalizacji THEN
	xAutonomizacja := TRUE;
END_IF 

// Kontrola komunikacji
fbTimerBrakuKomunikacji(IN := arModbusStatusKomunikacji[bAdres] = enumModbusStatus.BrakKomunikacji, PT := T#60S);
IF fbTimerBrakuKomunikacji.Q THEN
	xBrakKomunikacjiPLC := TRUE;
ELSE
	xBrakKomunikacjiPLC := FALSE;
END_IF

IF xAutonomizacja THEN
	xBrakKomunikacjiIZE := TRUE;
ELSE
	xBrakKomunikacjiIZE := FALSE;
END_IF

IF xPierwszySkan THEN
	xPierwszySkan := FALSE;
	WHILE arModbusOdczytCykliczny[intPetlaPierwszySkan].bAdresUrzadzenia <> 0 DO
		intPetlaPierwszySkan := intPetlaPierwszySkan + 1;
	END_WHILE

//deklaracja rejestrow do odczytu
	arModbusOdczytCykliczny[intPetlaPierwszySkan].bAdresUrzadzenia := bAdres;
	arModbusOdczytCykliczny[intPetlaPierwszySkan].bFunkcja := TO_BYTE(enumModbusKodyFunkcji.OdczytNRejestrow);
	arModbusOdczytCykliczny[intPetlaPierwszySkan].uiAdresRejestru := 50512;
	arModbusOdczytCykliczny[intPetlaPierwszySkan].ltCzestotliwosc := TIME_TO_LTIME(tMaksymalnyCzasRaportowania);
	arModbusOdczytCykliczny[intPetlaPierwszySkan].pZmiennaReferencyjna := ADR(wCzasPracyAnalizatoraHi);
	intPetlaPierwszySkan := intPetlaPierwszySkan + 1;

	arModbusOdczytCykliczny[intPetlaPierwszySkan].bAdresUrzadzenia := bAdres;
	arModbusOdczytCykliczny[intPetlaPierwszySkan].bFunkcja := TO_BYTE(enumModbusKodyFunkcji.OdczytNRejestrow);
	arModbusOdczytCykliczny[intPetlaPierwszySkan].uiAdresRejestru := 50513;
	arModbusOdczytCykliczny[intPetlaPierwszySkan].ltCzestotliwosc := TIME_TO_LTIME(tMaksymalnyCzasRaportowania);
	arModbusOdczytCykliczny[intPetlaPierwszySkan].pZmiennaReferencyjna := ADR(wCzasPracyAnalizatoraLo);
	intPetlaPierwszySkan := intPetlaPierwszySkan + 1;

	arModbusOdczytCykliczny[intPetlaPierwszySkan].bAdresUrzadzenia := bAdres;
	arModbusOdczytCykliczny[intPetlaPierwszySkan].bFunkcja := TO_BYTE(enumModbusKodyFunkcji.OdczytNRejestrow);
	arModbusOdczytCykliczny[intPetlaPierwszySkan].uiAdresRejestru := 50514;
	arModbusOdczytCykliczny[intPetlaPierwszySkan].ltCzestotliwosc := TIME_TO_LTIME(tMinimalnyCzasRaportowania);
	arModbusOdczytCykliczny[intPetlaPierwszySkan].pZmiennaReferencyjna := ADR(wNapiecieL1L2Hi);
	intPetlaPierwszySkan := intPetlaPierwszySkan + 1;

	arModbusOdczytCykliczny[intPetlaPierwszySkan].bAdresUrzadzenia := bAdres;
	arModbusOdczytCykliczny[intPetlaPierwszySkan].bFunkcja := TO_BYTE(enumModbusKodyFunkcji.OdczytNRejestrow);
	arModbusOdczytCykliczny[intPetlaPierwszySkan].uiAdresRejestru := 50515;
	arModbusOdczytCykliczny[intPetlaPierwszySkan].ltCzestotliwosc := TIME_TO_LTIME(tMinimalnyCzasRaportowania);
	arModbusOdczytCykliczny[intPetlaPierwszySkan].pZmiennaReferencyjna := ADR(wNapiecieL1L2Lo);
	intPetlaPierwszySkan := intPetlaPierwszySkan + 1;

	arModbusOdczytCykliczny[intPetlaPierwszySkan].bAdresUrzadzenia := bAdres;
	arModbusOdczytCykliczny[intPetlaPierwszySkan].bFunkcja := TO_BYTE(enumModbusKodyFunkcji.OdczytNRejestrow);
	arModbusOdczytCykliczny[intPetlaPierwszySkan].uiAdresRejestru := 50516;
	arModbusOdczytCykliczny[intPetlaPierwszySkan].ltCzestotliwosc := TIME_TO_LTIME(tMinimalnyCzasRaportowania);
	arModbusOdczytCykliczny[intPetlaPierwszySkan].pZmiennaReferencyjna := ADR(wNapiecieL2L3Hi);
	intPetlaPierwszySkan := intPetlaPierwszySkan + 1;
	
	arModbusOdczytCykliczny[intPetlaPierwszySkan].bAdresUrzadzenia := bAdres;
	arModbusOdczytCykliczny[intPetlaPierwszySkan].bFunkcja := TO_BYTE(enumModbusKodyFunkcji.OdczytNRejestrow);
	arModbusOdczytCykliczny[intPetlaPierwszySkan].uiAdresRejestru := 50517;
	arModbusOdczytCykliczny[intPetlaPierwszySkan].ltCzestotliwosc := TIME_TO_LTIME(tMinimalnyCzasRaportowania);
	arModbusOdczytCykliczny[intPetlaPierwszySkan].pZmiennaReferencyjna := ADR(wNapiecieL2L3Lo);
	intPetlaPierwszySkan := intPetlaPierwszySkan + 1;

	arModbusOdczytCykliczny[intPetlaPierwszySkan].bAdresUrzadzenia := bAdres;
	arModbusOdczytCykliczny[intPetlaPierwszySkan].bFunkcja := TO_BYTE(enumModbusKodyFunkcji.OdczytNRejestrow);
	arModbusOdczytCykliczny[intPetlaPierwszySkan].uiAdresRejestru := 50518;
	arModbusOdczytCykliczny[intPetlaPierwszySkan].ltCzestotliwosc := TIME_TO_LTIME(tMinimalnyCzasRaportowania);
	arModbusOdczytCykliczny[intPetlaPierwszySkan].pZmiennaReferencyjna := ADR(wNapiecieL3L1Hi);
	intPetlaPierwszySkan := intPetlaPierwszySkan + 1;
	
	arModbusOdczytCykliczny[intPetlaPierwszySkan].bAdresUrzadzenia := bAdres;
	arModbusOdczytCykliczny[intPetlaPierwszySkan].bFunkcja := TO_BYTE(enumModbusKodyFunkcji.OdczytNRejestrow);
	arModbusOdczytCykliczny[intPetlaPierwszySkan].uiAdresRejestru := 50519;
	arModbusOdczytCykliczny[intPetlaPierwszySkan].ltCzestotliwosc := TIME_TO_LTIME(tMinimalnyCzasRaportowania);
	arModbusOdczytCykliczny[intPetlaPierwszySkan].pZmiennaReferencyjna := ADR(wNapiecieL3L1Lo);
	intPetlaPierwszySkan := intPetlaPierwszySkan + 1;

	arModbusOdczytCykliczny[intPetlaPierwszySkan].bAdresUrzadzenia := bAdres;
	arModbusOdczytCykliczny[intPetlaPierwszySkan].bFunkcja := TO_BYTE(enumModbusKodyFunkcji.OdczytNRejestrow);
	arModbusOdczytCykliczny[intPetlaPierwszySkan].uiAdresRejestru := 50520;
	arModbusOdczytCykliczny[intPetlaPierwszySkan].ltCzestotliwosc := TIME_TO_LTIME(tMinimalnyCzasRaportowania);
	arModbusOdczytCykliczny[intPetlaPierwszySkan].pZmiennaReferencyjna := ADR(wNapiecieL1Hi);
	intPetlaPierwszySkan := intPetlaPierwszySkan + 1;

	arModbusOdczytCykliczny[intPetlaPierwszySkan].bAdresUrzadzenia := bAdres;
	arModbusOdczytCykliczny[intPetlaPierwszySkan].bFunkcja := TO_BYTE(enumModbusKodyFunkcji.OdczytNRejestrow);
	arModbusOdczytCykliczny[intPetlaPierwszySkan].uiAdresRejestru := 50521;
	arModbusOdczytCykliczny[intPetlaPierwszySkan].ltCzestotliwosc := TIME_TO_LTIME(tMinimalnyCzasRaportowania);
	arModbusOdczytCykliczny[intPetlaPierwszySkan].pZmiennaReferencyjna := ADR(wNapiecieL1Lo);
	intPetlaPierwszySkan := intPetlaPierwszySkan + 1;

	arModbusOdczytCykliczny[intPetlaPierwszySkan].bAdresUrzadzenia := bAdres;
	arModbusOdczytCykliczny[intPetlaPierwszySkan].bFunkcja := TO_BYTE(enumModbusKodyFunkcji.OdczytNRejestrow);
	arModbusOdczytCykliczny[intPetlaPierwszySkan].uiAdresRejestru := 50522;
	arModbusOdczytCykliczny[intPetlaPierwszySkan].ltCzestotliwosc := TIME_TO_LTIME(tMinimalnyCzasRaportowania);
	arModbusOdczytCykliczny[intPetlaPierwszySkan].pZmiennaReferencyjna := ADR(wNapiecieL2Hi);
	intPetlaPierwszySkan := intPetlaPierwszySkan + 1;
	
	arModbusOdczytCykliczny[intPetlaPierwszySkan].bAdresUrzadzenia := bAdres;
	arModbusOdczytCykliczny[intPetlaPierwszySkan].bFunkcja := TO_BYTE(enumModbusKodyFunkcji.OdczytNRejestrow);
	arModbusOdczytCykliczny[intPetlaPierwszySkan].uiAdresRejestru := 50523;
	arModbusOdczytCykliczny[intPetlaPierwszySkan].ltCzestotliwosc := TIME_TO_LTIME(tMinimalnyCzasRaportowania);
	arModbusOdczytCykliczny[intPetlaPierwszySkan].pZmiennaReferencyjna := ADR(wNapiecieL2Lo);
	intPetlaPierwszySkan := intPetlaPierwszySkan + 1;

	arModbusOdczytCykliczny[intPetlaPierwszySkan].bAdresUrzadzenia := bAdres;
	arModbusOdczytCykliczny[intPetlaPierwszySkan].bFunkcja := TO_BYTE(enumModbusKodyFunkcji.OdczytNRejestrow);
	arModbusOdczytCykliczny[intPetlaPierwszySkan].uiAdresRejestru := 50524;
	arModbusOdczytCykliczny[intPetlaPierwszySkan].ltCzestotliwosc := TIME_TO_LTIME(tMinimalnyCzasRaportowania);
	arModbusOdczytCykliczny[intPetlaPierwszySkan].pZmiennaReferencyjna := ADR(wNapiecieL3Hi);
	intPetlaPierwszySkan := intPetlaPierwszySkan + 1;
	
	arModbusOdczytCykliczny[intPetlaPierwszySkan].bAdresUrzadzenia := bAdres;
	arModbusOdczytCykliczny[intPetlaPierwszySkan].bFunkcja := TO_BYTE(enumModbusKodyFunkcji.OdczytNRejestrow);
	arModbusOdczytCykliczny[intPetlaPierwszySkan].uiAdresRejestru := 50525;
	arModbusOdczytCykliczny[intPetlaPierwszySkan].ltCzestotliwosc := TIME_TO_LTIME(tMinimalnyCzasRaportowania);
	arModbusOdczytCykliczny[intPetlaPierwszySkan].pZmiennaReferencyjna := ADR(wNapiecieL3Lo);
	intPetlaPierwszySkan := intPetlaPierwszySkan + 1;

	arModbusOdczytCykliczny[intPetlaPierwszySkan].bAdresUrzadzenia := bAdres;
	arModbusOdczytCykliczny[intPetlaPierwszySkan].bFunkcja := TO_BYTE(enumModbusKodyFunkcji.OdczytNRejestrow);
	arModbusOdczytCykliczny[intPetlaPierwszySkan].uiAdresRejestru := 50526;
	arModbusOdczytCykliczny[intPetlaPierwszySkan].ltCzestotliwosc := TIME_TO_LTIME(tMinimalnyCzasRaportowania);
	arModbusOdczytCykliczny[intPetlaPierwszySkan].pZmiennaReferencyjna := ADR(wCzestotliwoscHi);
	intPetlaPierwszySkan := intPetlaPierwszySkan + 1;

	arModbusOdczytCykliczny[intPetlaPierwszySkan].bAdresUrzadzenia := bAdres;
	arModbusOdczytCykliczny[intPetlaPierwszySkan].bFunkcja := TO_BYTE(enumModbusKodyFunkcji.OdczytNRejestrow);
	arModbusOdczytCykliczny[intPetlaPierwszySkan].uiAdresRejestru := 50527;
	arModbusOdczytCykliczny[intPetlaPierwszySkan].ltCzestotliwosc := TIME_TO_LTIME(tMinimalnyCzasRaportowania);
	arModbusOdczytCykliczny[intPetlaPierwszySkan].pZmiennaReferencyjna := ADR(wCzestotliwoscLo);
	intPetlaPierwszySkan := intPetlaPierwszySkan + 1;

	arModbusOdczytCykliczny[intPetlaPierwszySkan].bAdresUrzadzenia := bAdres;
	arModbusOdczytCykliczny[intPetlaPierwszySkan].bFunkcja := TO_BYTE(enumModbusKodyFunkcji.OdczytNRejestrow);
	arModbusOdczytCykliczny[intPetlaPierwszySkan].uiAdresRejestru := 50528;
	arModbusOdczytCykliczny[intPetlaPierwszySkan].ltCzestotliwosc := TIME_TO_LTIME(tMinimalnyCzasRaportowania);
	arModbusOdczytCykliczny[intPetlaPierwszySkan].pZmiennaReferencyjna := ADR(wPradL1Hi);
	intPetlaPierwszySkan := intPetlaPierwszySkan + 1;

	arModbusOdczytCykliczny[intPetlaPierwszySkan].bAdresUrzadzenia := bAdres;
	arModbusOdczytCykliczny[intPetlaPierwszySkan].bFunkcja := TO_BYTE(enumModbusKodyFunkcji.OdczytNRejestrow);
	arModbusOdczytCykliczny[intPetlaPierwszySkan].uiAdresRejestru := 50529;
	arModbusOdczytCykliczny[intPetlaPierwszySkan].ltCzestotliwosc := TIME_TO_LTIME(tMinimalnyCzasRaportowania);
	arModbusOdczytCykliczny[intPetlaPierwszySkan].pZmiennaReferencyjna := ADR(wPradL1Lo);
	intPetlaPierwszySkan := intPetlaPierwszySkan + 1;

	arModbusOdczytCykliczny[intPetlaPierwszySkan].bAdresUrzadzenia := bAdres;
	arModbusOdczytCykliczny[intPetlaPierwszySkan].bFunkcja := TO_BYTE(enumModbusKodyFunkcji.OdczytNRejestrow);
	arModbusOdczytCykliczny[intPetlaPierwszySkan].uiAdresRejestru := 50530;
	arModbusOdczytCykliczny[intPetlaPierwszySkan].ltCzestotliwosc := TIME_TO_LTIME(tMinimalnyCzasRaportowania);
	arModbusOdczytCykliczny[intPetlaPierwszySkan].pZmiennaReferencyjna := ADR(wPradL2Hi);
	intPetlaPierwszySkan := intPetlaPierwszySkan + 1;

	arModbusOdczytCykliczny[intPetlaPierwszySkan].bAdresUrzadzenia := bAdres;
	arModbusOdczytCykliczny[intPetlaPierwszySkan].bFunkcja := TO_BYTE(enumModbusKodyFunkcji.OdczytNRejestrow);
	arModbusOdczytCykliczny[intPetlaPierwszySkan].uiAdresRejestru := 50531;
	arModbusOdczytCykliczny[intPetlaPierwszySkan].ltCzestotliwosc := TIME_TO_LTIME(tMinimalnyCzasRaportowania);
	arModbusOdczytCykliczny[intPetlaPierwszySkan].pZmiennaReferencyjna := ADR(wPradL2Lo);
	intPetlaPierwszySkan := intPetlaPierwszySkan + 1;

	arModbusOdczytCykliczny[intPetlaPierwszySkan].bAdresUrzadzenia := bAdres;
	arModbusOdczytCykliczny[intPetlaPierwszySkan].bFunkcja := TO_BYTE(enumModbusKodyFunkcji.OdczytNRejestrow);
	arModbusOdczytCykliczny[intPetlaPierwszySkan].uiAdresRejestru := 50532;
	arModbusOdczytCykliczny[intPetlaPierwszySkan].ltCzestotliwosc := TIME_TO_LTIME(tMinimalnyCzasRaportowania);
	arModbusOdczytCykliczny[intPetlaPierwszySkan].pZmiennaReferencyjna := ADR(wPradL3Hi);
	intPetlaPierwszySkan := intPetlaPierwszySkan + 1;

	arModbusOdczytCykliczny[intPetlaPierwszySkan].bAdresUrzadzenia := bAdres;
	arModbusOdczytCykliczny[intPetlaPierwszySkan].bFunkcja := TO_BYTE(enumModbusKodyFunkcji.OdczytNRejestrow);
	arModbusOdczytCykliczny[intPetlaPierwszySkan].uiAdresRejestru := 50533;
	arModbusOdczytCykliczny[intPetlaPierwszySkan].ltCzestotliwosc := TIME_TO_LTIME(tMinimalnyCzasRaportowania);
	arModbusOdczytCykliczny[intPetlaPierwszySkan].pZmiennaReferencyjna := ADR(wPradL3Lo);
	intPetlaPierwszySkan := intPetlaPierwszySkan + 1;

	arModbusOdczytCykliczny[intPetlaPierwszySkan].bAdresUrzadzenia := bAdres;
	arModbusOdczytCykliczny[intPetlaPierwszySkan].bFunkcja := TO_BYTE(enumModbusKodyFunkcji.OdczytNRejestrow);
	arModbusOdczytCykliczny[intPetlaPierwszySkan].uiAdresRejestru := 50534;
	arModbusOdczytCykliczny[intPetlaPierwszySkan].ltCzestotliwosc := TIME_TO_LTIME(tMinimalnyCzasRaportowania);
	arModbusOdczytCykliczny[intPetlaPierwszySkan].pZmiennaReferencyjna := ADR(wPradNHi);
	intPetlaPierwszySkan := intPetlaPierwszySkan + 1;

	arModbusOdczytCykliczny[intPetlaPierwszySkan].bAdresUrzadzenia := bAdres;
	arModbusOdczytCykliczny[intPetlaPierwszySkan].bFunkcja := TO_BYTE(enumModbusKodyFunkcji.OdczytNRejestrow);
	arModbusOdczytCykliczny[intPetlaPierwszySkan].uiAdresRejestru := 50535;
	arModbusOdczytCykliczny[intPetlaPierwszySkan].ltCzestotliwosc := TIME_TO_LTIME(tMinimalnyCzasRaportowania);
	arModbusOdczytCykliczny[intPetlaPierwszySkan].pZmiennaReferencyjna := ADR(wPradNLo);
	intPetlaPierwszySkan := intPetlaPierwszySkan + 1;
	
	arModbusOdczytCykliczny[intPetlaPierwszySkan].bAdresUrzadzenia := bAdres;
	arModbusOdczytCykliczny[intPetlaPierwszySkan].bFunkcja := TO_BYTE(enumModbusKodyFunkcji.OdczytNRejestrow);
	arModbusOdczytCykliczny[intPetlaPierwszySkan].uiAdresRejestru := 50536;
	arModbusOdczytCykliczny[intPetlaPierwszySkan].ltCzestotliwosc := TIME_TO_LTIME(tMinimalnyCzasRaportowania);
	arModbusOdczytCykliczny[intPetlaPierwszySkan].pZmiennaReferencyjna := ADR(wMocCzynnaCalkowitaHi);
	intPetlaPierwszySkan := intPetlaPierwszySkan + 1;
	
	arModbusOdczytCykliczny[intPetlaPierwszySkan].bAdresUrzadzenia := bAdres;
	arModbusOdczytCykliczny[intPetlaPierwszySkan].bFunkcja := TO_BYTE(enumModbusKodyFunkcji.OdczytNRejestrow);
	arModbusOdczytCykliczny[intPetlaPierwszySkan].uiAdresRejestru := 50537;
	arModbusOdczytCykliczny[intPetlaPierwszySkan].ltCzestotliwosc := TIME_TO_LTIME(tMinimalnyCzasRaportowania);
	arModbusOdczytCykliczny[intPetlaPierwszySkan].pZmiennaReferencyjna := ADR(wMocCzynnaCalkowitaLo);
	intPetlaPierwszySkan := intPetlaPierwszySkan + 1;
	
	arModbusOdczytCykliczny[intPetlaPierwszySkan].bAdresUrzadzenia := bAdres;
	arModbusOdczytCykliczny[intPetlaPierwszySkan].bFunkcja := TO_BYTE(enumModbusKodyFunkcji.OdczytNRejestrow);
	arModbusOdczytCykliczny[intPetlaPierwszySkan].uiAdresRejestru := 50538;
	arModbusOdczytCykliczny[intPetlaPierwszySkan].ltCzestotliwosc := TIME_TO_LTIME(tMinimalnyCzasRaportowania);
	arModbusOdczytCykliczny[intPetlaPierwszySkan].pZmiennaReferencyjna := ADR(wMocBiernaCalkowitaHi);
	intPetlaPierwszySkan := intPetlaPierwszySkan + 1;
	
	arModbusOdczytCykliczny[intPetlaPierwszySkan].bAdresUrzadzenia := bAdres;
	arModbusOdczytCykliczny[intPetlaPierwszySkan].bFunkcja := TO_BYTE(enumModbusKodyFunkcji.OdczytNRejestrow);
	arModbusOdczytCykliczny[intPetlaPierwszySkan].uiAdresRejestru := 50539;
	arModbusOdczytCykliczny[intPetlaPierwszySkan].ltCzestotliwosc := TIME_TO_LTIME(tMinimalnyCzasRaportowania);
	arModbusOdczytCykliczny[intPetlaPierwszySkan].pZmiennaReferencyjna := ADR(wMocBiernaCalkowitaLo);
	intPetlaPierwszySkan := intPetlaPierwszySkan + 1;
	
	arModbusOdczytCykliczny[intPetlaPierwszySkan].bAdresUrzadzenia := bAdres;
	arModbusOdczytCykliczny[intPetlaPierwszySkan].bFunkcja := TO_BYTE(enumModbusKodyFunkcji.OdczytNRejestrow);
	arModbusOdczytCykliczny[intPetlaPierwszySkan].uiAdresRejestru := 50540;
	arModbusOdczytCykliczny[intPetlaPierwszySkan].ltCzestotliwosc := TIME_TO_LTIME(tMinimalnyCzasRaportowania);
	arModbusOdczytCykliczny[intPetlaPierwszySkan].pZmiennaReferencyjna := ADR(wMocPozornaCalkowitaHi);
	intPetlaPierwszySkan := intPetlaPierwszySkan + 1;
	
	arModbusOdczytCykliczny[intPetlaPierwszySkan].bAdresUrzadzenia := bAdres;
	arModbusOdczytCykliczny[intPetlaPierwszySkan].bFunkcja := TO_BYTE(enumModbusKodyFunkcji.OdczytNRejestrow);
	arModbusOdczytCykliczny[intPetlaPierwszySkan].uiAdresRejestru := 50541;
	arModbusOdczytCykliczny[intPetlaPierwszySkan].ltCzestotliwosc := TIME_TO_LTIME(tMinimalnyCzasRaportowania);
	arModbusOdczytCykliczny[intPetlaPierwszySkan].pZmiennaReferencyjna := ADR(wMocPozornaCalkowitaLo);
	intPetlaPierwszySkan := intPetlaPierwszySkan + 1;
	
	arModbusOdczytCykliczny[intPetlaPierwszySkan].bAdresUrzadzenia := bAdres;
	arModbusOdczytCykliczny[intPetlaPierwszySkan].bFunkcja := TO_BYTE(enumModbusKodyFunkcji.OdczytNRejestrow);
	arModbusOdczytCykliczny[intPetlaPierwszySkan].uiAdresRejestru := 50542;
	arModbusOdczytCykliczny[intPetlaPierwszySkan].ltCzestotliwosc := TIME_TO_LTIME(tMinimalnyCzasRaportowania);
	arModbusOdczytCykliczny[intPetlaPierwszySkan].pZmiennaReferencyjna := ADR(wWspolczynnikMocyCalkowityHi);
	intPetlaPierwszySkan := intPetlaPierwszySkan + 1;
	
	arModbusOdczytCykliczny[intPetlaPierwszySkan].bAdresUrzadzenia := bAdres;
	arModbusOdczytCykliczny[intPetlaPierwszySkan].bFunkcja := TO_BYTE(enumModbusKodyFunkcji.OdczytNRejestrow);
	arModbusOdczytCykliczny[intPetlaPierwszySkan].uiAdresRejestru := 50543;
	arModbusOdczytCykliczny[intPetlaPierwszySkan].ltCzestotliwosc := TIME_TO_LTIME(tMinimalnyCzasRaportowania);
	arModbusOdczytCykliczny[intPetlaPierwszySkan].pZmiennaReferencyjna := ADR(wWspolczynnikMocyCalkowityLo);
	intPetlaPierwszySkan := intPetlaPierwszySkan + 1;

	arModbusOdczytCykliczny[intPetlaPierwszySkan].bAdresUrzadzenia := bAdres;
	arModbusOdczytCykliczny[intPetlaPierwszySkan].bFunkcja := TO_BYTE(enumModbusKodyFunkcji.OdczytNRejestrow);
	arModbusOdczytCykliczny[intPetlaPierwszySkan].uiAdresRejestru := 50554;
	arModbusOdczytCykliczny[intPetlaPierwszySkan].ltCzestotliwosc := TIME_TO_LTIME(tMinimalnyCzasRaportowania);
	arModbusOdczytCykliczny[intPetlaPierwszySkan].pZmiennaReferencyjna := ADR(wMocBiernaL3Hi);
	intPetlaPierwszySkan := intPetlaPierwszySkan + 1;

	arModbusOdczytCykliczny[intPetlaPierwszySkan].bAdresUrzadzenia := bAdres;
	arModbusOdczytCykliczny[intPetlaPierwszySkan].bFunkcja := TO_BYTE(enumModbusKodyFunkcji.OdczytNRejestrow);
	arModbusOdczytCykliczny[intPetlaPierwszySkan].uiAdresRejestru := 50555;
	arModbusOdczytCykliczny[intPetlaPierwszySkan].ltCzestotliwosc := TIME_TO_LTIME(tMinimalnyCzasRaportowania);
	arModbusOdczytCykliczny[intPetlaPierwszySkan].pZmiennaReferencyjna := ADR(wMocBiernaL3Lo);
	intPetlaPierwszySkan := intPetlaPierwszySkan + 1;
	
	arModbusOdczytCykliczny[intPetlaPierwszySkan].bAdresUrzadzenia := bAdres;
	arModbusOdczytCykliczny[intPetlaPierwszySkan].bFunkcja := TO_BYTE(enumModbusKodyFunkcji.OdczytNRejestrow);
	arModbusOdczytCykliczny[intPetlaPierwszySkan].uiAdresRejestru := 50552;
	arModbusOdczytCykliczny[intPetlaPierwszySkan].ltCzestotliwosc := TIME_TO_LTIME(tMinimalnyCzasRaportowania);
	arModbusOdczytCykliczny[intPetlaPierwszySkan].pZmiennaReferencyjna := ADR(wMocBiernaL2Hi);
	intPetlaPierwszySkan := intPetlaPierwszySkan + 1;

	arModbusOdczytCykliczny[intPetlaPierwszySkan].bAdresUrzadzenia := bAdres;
	arModbusOdczytCykliczny[intPetlaPierwszySkan].bFunkcja := TO_BYTE(enumModbusKodyFunkcji.OdczytNRejestrow);
	arModbusOdczytCykliczny[intPetlaPierwszySkan].uiAdresRejestru := 50553;
	arModbusOdczytCykliczny[intPetlaPierwszySkan].ltCzestotliwosc := TIME_TO_LTIME(tMinimalnyCzasRaportowania);
	arModbusOdczytCykliczny[intPetlaPierwszySkan].pZmiennaReferencyjna := ADR(wMocBiernaL2Lo);
	intPetlaPierwszySkan := intPetlaPierwszySkan + 1;	
	
	arModbusOdczytCykliczny[intPetlaPierwszySkan].bAdresUrzadzenia := bAdres;
	arModbusOdczytCykliczny[intPetlaPierwszySkan].bFunkcja := TO_BYTE(enumModbusKodyFunkcji.OdczytNRejestrow);
	arModbusOdczytCykliczny[intPetlaPierwszySkan].uiAdresRejestru := 50550;
	arModbusOdczytCykliczny[intPetlaPierwszySkan].ltCzestotliwosc := TIME_TO_LTIME(tMinimalnyCzasRaportowania);
	arModbusOdczytCykliczny[intPetlaPierwszySkan].pZmiennaReferencyjna := ADR(wMocBiernaL1Hi);
	intPetlaPierwszySkan := intPetlaPierwszySkan + 1;

	arModbusOdczytCykliczny[intPetlaPierwszySkan].bAdresUrzadzenia := bAdres;
	arModbusOdczytCykliczny[intPetlaPierwszySkan].bFunkcja := TO_BYTE(enumModbusKodyFunkcji.OdczytNRejestrow);
	arModbusOdczytCykliczny[intPetlaPierwszySkan].uiAdresRejestru := 50551;
	arModbusOdczytCykliczny[intPetlaPierwszySkan].ltCzestotliwosc := TIME_TO_LTIME(tMinimalnyCzasRaportowania);
	arModbusOdczytCykliczny[intPetlaPierwszySkan].pZmiennaReferencyjna := ADR(wMocBiernaL1Lo);
	intPetlaPierwszySkan := intPetlaPierwszySkan + 1;	


